# B&R Automation Studio project Soiled_PLC (part 2)

#### zzbagsfl.ab
```automation-basic
PROGRAM _CYCLIC

;----------------------------------------------------------------------
;Version 1.00 19/12/2005 D.J. First Issue - Using BAG array
;Version 2.00 24/06/2009 D.J. 32bit Cat and Cus .Cat replaced with .Prg
;Version 3.00 09/11/2009 D.J. Added Destination Counts
;----------------------------------------------------------------------
;***************************************ZEROSPOT SPECIAL*****************
Std.BagsWithDestinations 	= FALSE
Std.CustomerFound	 		   = FALSE
Std.BagsWithDestinations2  = FALSE

;Clear Destination Counts
memset(ADR(DestCountStorage),0,SIZEOF(DestCountStorage))
memset(ADR(DestCountSystem),0,SIZEOF(DestCountSystem))

LOOP CurrentLine = 1 to Std.MaxLinesBuffers DO

	LineSp = 0

	LOOP CurrentBag = Line[CurrentLine].FirstBag  TO Line[CurrentLine].LastBag DO

		EXITIF Line[CurrentLine].FirstBag = 0

		NextBag = (CurrentBag + 1)

		IF ((CurrentBag < Line[CurrentLine].LastBag) AND ((Bag[CurrentBag].Cat = 0) AND (Bag[NextBag].Cat > 0))) THEN

			;Copy Next Bag to Current
			Bag[CurrentBag]	= Bag[NextBag]
			Bag[NextBag] 	= Bag[0]

		ENDIF

		;Speed up task buy using simple variables saved 0.5ms from this task 5% CPU Usage
		CurrentDst		= Bag[CurrentBag].Dst
		IF ((CurrentDst > 0) AND (CurrentDst <= MAX_DESTINATIONS)) THEN
			IF (CurrentLine <= Std.MaxLines) THEN
				Std.BagsWithDestinations = TRUE
				DestCountStorage[CurrentDst] = DestCountStorage[CurrentDst] + 1
			ENDIF
;			DestCountSystem[CurrentDst] = DestCountSystem[CurrentDst] + 1
		ELSE IF (CurrentDst > MAX_DESTINATIONS)THEN
			Bag[CurrentBag].Dst := 0;
		ELSE IF ((CurrentDst >0) AND (CurrentDst  <= MAX_DESTINATIONS) AND (CurrentLine = 30))	THEN
			;Std.BagsWithDestinations2 = TRUE
			;DestCountStorage[CurrentDst] = DestCountStorage[CurrentDst] + 1
		ENDIF
			;FOUL LOOP bag with destination
		IF ((CurrentDst >0) AND (CurrentDst  <= MAX_DESTINATIONS) AND (CurrentLine = 30))	THEN
			Std.BagsWithDestinations2 = TRUE
			DestCountStorage[CurrentDst] = DestCountStorage[CurrentDst] + 1
		ENDIF
		;Add the line spaces up
		IF Bag[CurrentBag].Cat = 0 THEN
			LineSp = (LineSp + 1)
		ENDIF

		;For Customer FIFO table
		;-----------------------
		;Customer at front of FIFO in Storage
		;****************SPECIAL FOR ZEROSPOT*******************************
		IF ((Bag[CurrentBag].Cus = D32[401]) AND (D32[401] > 0) AND (CurrentLine <= Std.MaxLines)) THEN
			Std.CustomerFound	 	= TRUE
		ENDIF
		//Special for pairing loop, do not delete custmoer from FIFO if its on the loop
		IF ((Bag[CurrentBag].Cus = D32[401]) AND (D32[401] > 0) AND ((CurrentLine >= 30) OR (CurrentLine <= 32))) THEN
			Std.CustomerFound	 	= TRUE
		ENDIF
		IF ((Bag[259].Cus = D32[401]) AND (D32[401] > 0)) THEN
			Std.CustomerFound	 	= TRUE
		ENDIF

	ENDLOOP
	;Save the number of spaces on the current line
	Line[CurrentLine].Space = LineSp

ENDLOOP
IF (Bag[151].Cat = 0) THEN
	Line[19].Space = Line[19].Space + 1
ENDIF

IF (Bag[157].Cat = 0) THEN
	Line[19].Space = Line[19].Space + 1
ENDIF

END_PROGRAM
```

### Program Logical/Sequences/10ms/zzcp10ser (IEC, version 3.00.1)

#### zzstnser.var
```iecst
VAR
	MixProgTyp : BOOL;
	BatchFound : BOOL;
	MixCusts : BOOL;
	MixProgs : BOOL;
	MatchCust : BOOL;
	MatchBags : BOOL;
	MatchProgType : BOOL;
	MatchProg : BOOL;
	MatchCat : BOOL;
	StartPurge : BOOL;
	MixCats : BOOL;
	BankValid : BOOL;
	LineValid : BOOL;
	BagInList : ARRAY[0..30] OF BOOL;
	StartPurgeET : UDINT;
	BagNum : UINT;
	BagWgt : UINT;
	Index : UINT;
	PurgeBagsQty : UINT;
	StnNum : UINT;
	BatchCount : UINT;
	s : UINT;
	BatchWeight : UINT;
	myBag : UINT;
	r : UINT;
	MaxReverseWeight : UINT;
END_VAR
VAR RETAIN
	LineSearchManual : UINT;
END_VAR
VAR
	NumberOfPurgeBags : UINT;
	x : UINT;
END_VAR
VAR RETAIN
	SearchLine : UINT;
END_VAR
VAR
	Bank : UINT;
	Choice : UINT;
	EndofBagArray : UINT;
	PurgeBatchSize : UINT;
	MaxBatchWieght : UINT;
END_VAR
VAR RETAIN
	n : UINT;
END_VAR
VAR
	t : UINT;
	myBag_x : UINT;
	myBag_n : UINT;
END_VAR
VAR RETAIN
	SearchFound : UINT;
END_VAR
VAR
	LineSearch : ARRAY[0..4] OF UINT;
	SearchBagArray : ARRAY[0..30] OF UINT;
	PurgeBags : ARRAY[0..30] OF UINT;
	PurgeBagsInWgtOrder : ARRAY[0..30] OF UINT;
	PurgeOn : UINT;
	StatusReg : ARRAY[0..1] OF UDINT;
	SearchIndex : USINT;
	ReSearch : BOOL;
	MisMatchedLoad : BOOL;
	y : INT;
	Break : BOOL;
	StnCat : UDINT;
	GetStn : UINT;
	TestTim : BOOL;
	myStartStop : UINT;
	b : UINT;
	TON_Purge : ARRAY[0..4] OF TON_10ms;
	myBatchWgt : UDINT;
	test : UDINT;
	EmptyViking : ARRAY[0..20] OF BOOL;
	Priority : ARRAY[0..20] OF BOOL;
	E : BOOL;
	Normal : UINT;
	Over1 : UINT;
	Over2 : UINT;
	Over3 : UINT;
	Over4 : UINT;
	Viking : ARRAY[0..20] OF USINT;
	Dest : UINT;
END_VAR
```

#### zzstnser.ab
```automation-basic
;-----------------------------------------------------
;Sorting Station Search Routine - No changes required!
;-----------------------------------------------------

;----------------------------------------
;Version 1.00 19/12/2005 First Issue D.J.
;Version 2.00 03/11/2010 Revised D.J.
;Version 3.00 19/07/2016 TR... Fix bug so multiple banks can release whilst purging..
;----------------------------------------

PROGRAM _CYCLIC

IF Ldg[3].Search = 1 THEN

;Viking 5 CDC 5
IF ((Bag[80].Cat = 0) AND (Bag[81].Cat = 0) AND (Bag[82].Cat = 0)) THEN
	EmptyViking[15] = TRUE

ELSE IF ((Bag[81].Cat = 0 = 0) AND (Bag[82].Cat = 0)) THEN
	Priority[15] = TRUE

ELSE
	Priority[15]    = FALSE
	EmptyViking[15] = FALSE
ENDIF

;Viking 4 CDC 6
IF ((Bag[85].Cat = 0) AND (Bag[86].Cat = 0) AND (Bag[87].Cat = 0)) THEN
	EmptyViking[16] = TRUE

ELSE IF ((Bag[86].Cat = 0) AND (Bag[87].Cat = 0)) THEN
	Priority[16] = TRUE
ELSE
	Priority[16]    = FALSE
	EmptyViking[16] = FALSE
ENDIF

;Viking 3 CDC 7
IF ((Bag[90].Cat = 0) AND (Bag[91].Cat = 0) AND (Bag[92].Cat = 0)) THEN
	EmptyViking[16] = TRUE
ELSE IF ((Bag[91].Cat = 0) AND (Bag[92].Cat = 0)) THEN
	Priority[17] = TRUE
ELSE
	Priority[17]    = FALSE
	EmptyViking[17] = FALSE
ENDIF

;Viking 2 CDC 8
IF ((Bag[95].Cat = 0) AND (Bag[96].Cat = 0) AND (Bag[97].Cat = 0)) THEN
	EmptyViking[18] = TRUE
ELSE IF ((Bag[97].Cat = 0) AND (Bag[96].Cat = 0)) THEN
	Priority[18] = TRUE
ELSE
	Priority[18]    = FALSE
	EmptyViking[18] = FALSE
ENDIF

IF ((Bag[101].Cat = 0) AND (Bag[102].Cat = 0)AND (Bag[157].Cat = 0) AND (Bag[151].Cat = 0)) THEN
	EmptyViking[18] = TRUE
ELSE IF ((Bag[101].Cat = 0) AND (Bag[102].Cat = 0)AND (Bag[157].Cat = 0) AND (Bag[151].Cat = 0)) THEN
	Priority[19] = TRUE
ELSE
	Priority[19]    = FALSE
	EmptyViking[19] = FALSE
ENDIF

             n       = UINT(Bag[154].Cat)
      		 Normal  = (D[3000 + n]) ;destinations from cat data base
   	  		 Over1   = (D[3100 + n])
   	  		 Over2   = (D[3200 + n])
   	  		 Over3   = (D[3300 + n])
   	  		 ;Over4   = (D[2400 + n])

   	IF ((Line[Normal].SpaceBIT = 2 ) AND (D[Normal] = 1)AND (EmptyViking[Normal] = TRUE)) THEN
      	Dest = Normal
   ELSE IF ((Line[Over1].SpaceBIT = 2) AND (D[Over1] = 1 )AND (EmptyViking[Over1] = TRUE)) THEN
        Dest = Over1
   ELSE IF ((Line[Over2].SpaceBIT = 2 ) AND (D[Over2] = 1 )AND (EmptyViking[Over2] = TRUE)) THEN
        Dest = Over2
   ELSE IF ((Line[Over3].SpaceBIT = 2 ) AND (D[Over3] = 1 )AND (EmptyViking[Over3] = TRUE)) THEN
        Dest = Over3
   ;ELSE IF ((Viking[Over4] = 2 ) AND (D[Over4 ] = 1 )AND (EmptyViking[Over4] = TRUE)) THEN
    ;    Dest = Over4

   ELSE IF ((Line[Normal].SpaceBIT = 2 ) AND (D[Normal] = 1)AND (Priority[Normal] = TRUE)) THEN
      	Dest = Normal
   ELSE IF ((Line[Over1].SpaceBIT = 2) AND (D[Over1] = 1 )AND (Priority[Over1] = TRUE)) THEN
        Dest = Over1
   ELSE IF ((Line[Over2].SpaceBIT = 2 ) AND (D[Over2] = 1 )AND (Priority[Over2] = TRUE)) THEN
        Dest = Over2
   ELSE IF ((Line[Over3].SpaceBIT = 2 ) AND (D[Over3] = 1 )AND (Priority[Over3] = TRUE)) THEN
        Dest = Over3
   ;ELSE IF ((Viking[Over4] = 2 ) AND (D[Over4 + 7] = 1 )AND (Priority[Over4] = TRUE)) THEN
   ;     Dest = Over4
    ELSE IF ((Line[Normal].SpaceBIT > 0 ) AND (D[Normal ] = 1)) THEN
       Dest = Normal
    ELSE IF ((Line[Over1].SpaceBIT > 0) AND (D[Over1] = 1 )) THEN
        Dest = Over1
   ELSE IF ((Line[Over2].SpaceBIT > 0 ) AND (D[Over2] = 1 )) THEN
        Dest = Over2
   ELSE IF ((Line[Over3].SpaceBIT > 0 ) AND (D[Over3] = 1 )) THEN
        Dest = Over3
   ;ELSE IF ((Viking[Over4] > 0 ) AND (D[Over4 + 7] = 1 )) THEN
   ;     Dest = Over4
   ENDIF

  IF ((Dest > 0) AND (Bag[154].Dst = 0) AND (Line[Dest].SpaceBIT>0)) THEN
  	Ldg[3].Search = 2
  	Ldg[3].Found       = Dest
  ELSE IF (Bag[154].Dst > 14)AND (Line[Bag[154].Dst].SpaceBIT>0) THEN
  	Ldg[3].Search = 2
  	Ldg[3].Found       = Bag[154].Dst
 ENDIF
ENDIF
Debug:

END_PROGRAM
```

### Program Logical/Sequences/10ms/zzBITcal (IEC) - * Bags In Transit Calculation

#### zzbitcal.var
```iecst
VAR RETAIN
	TotalTransitBags : UINT;
	n : UINT;
	BITDest : ARRAY[0..199] OF UINT;
	Destination : USINT;
	SpaceBIT : ARRAY[0..199] OF UINT;
	Spaces : INT;
END_VAR
VAR
	BITBag : UINT;
	ArraySize : UINT;
	Error : UINT;
	BoostSD4 : BOOL;
	BoostSDC4 : BOOL;
	BoostSDC5 : BOOL;
	lineValid : BOOL;
END_VAR
```

#### zzbitcal.ab
```automation-basic
PROGRAM _INIT

BITBag 	= 2
Error 	= 0
;Transfer Belt Bags
;LOOP n = 1 TO 2 DO
	;BITDest[1] = 153
	;BITDest[2] = 152
	;BITDest[3] = 151
	;BITDest[4] = 157
;	BITDest[BITBag] = n
;	BITBag = BITBag + 1
;ENDLOOP

;Bags in transit
LOOP n = 110 TO 164 DO

	ArraySize = (SIZEOF(BITDest) / 2)
	IF (BITBag <= ArraySize) THEN
		BITDest[BITBag] = n
		BITBag = BITBag + 1
	ELSE
		Error = 1
	ENDIF
ENDLOOP

TotalTransitBags = (BITBag - 1)
END_PROGRAM

PROGRAM _CYCLIC
	(* cyclic program *)

	;-----------------------------------------------------------
	;Revision 1.00 19/12/2005 D.J. First Issue - Using BAG array
	;-----------------------------------------------------------

	;Find the Space on each Storage line including the Ongoing and Offgoing Bags In Transit

	;See Init Routine - Change settings for bags in transit bag numbers

	;Clear local calculation
	LOOP n = 1 TO Std.MaxLinesBuffers DO
		SpaceBIT[n] = 0
	ENDLOOP

	memset(ADR(DestCountArea1),0,SIZEOF(DestCountArea1))

	;Ensure the destination is less than the Array size of SpaceBIT	(normally 100)
	LOOP n = 1 TO TotalTransitBags DO
	;LOOP n = 3 TO 3 DO
		Destination = Bag[BITDest[n]].Dst

		lineValid = ((Destination <= Line[Destination].FirstBag) OR (Destination > Line[Destination].LastBag));//Stop bit being counted twice if on own line.
		IF lineValid AND (Destination > 0) AND (Destination < 15)  THEN
			SpaceBIT[Destination] = SpaceBIT[Destination] + 1
			DestCountSystem[Destination] = DestCountSystem[Destination] + 1
		ENDIF
	ENDLOOP
	IF (Bag[153].Cat > 0) AND (Bag[153].Dst>0) THEN
			SpaceBIT[Bag[153].Dst] = SpaceBIT[Bag[153].Dst] + 1
			DestCountSystem[Bag[153].Dst] = DestCountSystem[Bag[153].Dst] + 1
	ENDIF
	IF (Bag[152].Cat > 0) AND (Bag[152].Dst>0) THEN
			SpaceBIT[Bag[152].Dst] = SpaceBIT[Bag[152].Dst] + 1
			DestCountSystem[Bag[152].Dst] = DestCountSystem[Bag[152].Dst] + 1
	ENDIF
	IF (Bag[166].Cat > 0) AND (Bag[166].Dst>0) THEN
			SpaceBIT[Bag[166].Dst] = SpaceBIT[Bag[166].Dst] + 1
			DestCountSystem[Bag[166].Dst] = DestCountSystem[Bag[166].Dst] + 1
	ENDIF
	IF (Bag[151].Cat > 0) AND (Bag[151].Dst>0) THEN
			SpaceBIT[Bag[151].Dst] = SpaceBIT[Bag[151].Dst] + 1
			DestCountSystem[Bag[151].Dst] = DestCountSystem[Bag[151].Dst] + 1
	ENDIF
	IF (Bag[157].Cat > 0) AND (Bag[157].Dst>0) THEN
			SpaceBIT[Bag[157].Dst] = SpaceBIT[Bag[157].Dst] + 1
			DestCountSystem[Bag[157].Dst] = DestCountSystem[Bag[157].Dst] + 1
	ENDIF
	;Once all calculated then update the global line space
	LOOP n = 1 TO Std.MaxLinesBuffers DO
	;LOOP n = 1 TO 1 DO
		Spaces = (INT(Line[n].Space) - INT(SpaceBIT[n]))
		IF Spaces > 0 THEN
			Line[n].SpaceBIT = UINT(Spaces)
		ELSE
			Line[n].SpaceBIT = 0
		ENDIF
	ENDLOOP

END_PROGRAM
```

### Program Logical/Sequences/10ms/zzCusFIFO (IEC) - * Customer FIFO 

#### zcusfifo.var
```iecst
VAR RETAIN
	OngoingCus : UDINT;
	EditCus : UDINT;
	n : UDINT;
	x : UINT;
END_VAR
VAR
	myBag : UINT;
	InsDel : DINT;
	InsPos : UDINT;
	DelPos : UDINT;
END_VAR
```

#### zcusfifo.ab
```automation-basic
PROGRAM _CYCLIC
;------------------------------------------------------
;Revision 1.00 11/02/2002 D.J. First Issue
;Revision 2.00 11/06/2002 D.J. Included Bags In Transit
;------------------------------------------------------

;Include any Bags In Transit if required

;New Customers
InsPos		= D32[496]
DelPos		= D32[497]
OngoingCus 	= D32[498]
EditCus		= D32[499]

IF Std.CustomerFIFO THEN

	;The following are Set by the "Bag Shuffle"
	;First customer not found clear from the FIFO
	IF NOT Std.CustomerFound THEN
		D32[401] = 0
	ENDIF

	;Shuffle the Table down
	D32[400] = 0

	LOOP n = 401 TO 494 DO

		IF ((D32[n] = 0) AND (D32[n + 1] > 0)) THEN
			D32[n] = D32[n + 1]
			D32[n + 1] = 0
		ENDIF

		IF (D32[n] > 0) THEN
			;Inc FIFO Header Count
			D32[400] = (D32[400] + 1)
		ENDIF

		;Clear New Customer if found
		IF ((OngoingCus > 0) AND (OngoingCus = D32[n])) THEN
			OngoingCus = 0
		ENDIF

		;Clear Edited Customer if found
		IF ((EditCus > 0) AND (EditCus = D32[n])) THEN
			EditCus = 0
		ENDIF

	ENDLOOP

	;Insert From TrackView
	IF ((InsPos > 0) AND (EditCus > 0)) THEN
		LOOP n = 495 DOWNTO (400 + InsPos) DO
			D32[n] = D32[n - 1]
		ENDLOOP
		D32[400 + InsPos] 	= EditCus
		InsPos 				= 0
		EditCus				= 0
	ENDIF

	;Delets From TrackView
	IF (DelPos > 0) THEN
		D32[400 + DelPos] 	= 0
		DelPos 				= 0
	ENDIF

	;D32[498] = Ongoing New Customer
	IF ((OngoingCus > 0) AND (D32[401 + D32[400]] = 0)) THEN
		D32[401 + D32[400]]	= OngoingCus
		OngoingCus 			= 0
		D32[400] 			= (D32[400] + 1)
	ENDIF

	;D32[499] = Edited New Customer
	IF ((EditCus > 0) AND (D32[401 + D32[400]] = 0)) THEN
		D32[401 + D32[400]]	= EditCus
		EditCus 			= 0
		D32[400] 			= (D32[400] + 1)
	ENDIF

	;Find the Current Customer for each Discharger and allocate the Next Customer

	LOOP x = 1 TO Std.MaxDischargers DO

		Uld[x].FIFONextCustomer = 0
		Uld[x].FIFOCustomerFound = FALSE

		;If No Customer then Allocate with the First
		IF (Uld[x].FIFOCustomer = 0) THEN
			Uld[x].FIFOCustomer = D32[401]
		ENDIF

		;If Next Customer available then allocate New Customer
		IF (D32[400] > 0) THEN
			LOOP n = 401 TO (D32[400] + 400) DO
				IF ((Uld[x].FIFOCustomer = D32[n]) AND (D32[n] > 0)) THEN
					Uld[x].FIFOCustomerFound = TRUE
					IF (D32[n + 1] > 0) THEN
						Uld[x].FIFONextCustomer = D32[n + 1]
					ENDIF
				ENDIF
			ENDLOOP
		ENDIF

		;If the current customer has been removed then set the next as the first
		IF ((Uld[x].FIFONextCustomer = 0) AND NOT Uld[x].FIFOCustomerFound) THEN
			Uld[x].FIFONextCustomer = D32[401]
		ENDIF

	ENDLOOP

ENDIF

D32[496] = InsPos
D32[497] = DelPos
D32[498] = OngoingCus
D32[499] = EditCus
END_PROGRAM
```

- Program Logical/Sequences/10ms/zzCount (IEC) - Counting frames inputs & Piece Weights (no source held here)

### Program Logical/Sequences/10ms/zzStnMix (IEC)

#### zzstnmix.ab
```automation-basic
PROGRAM _CYCLIC
;----------------------
;Sorting Station Mixing
;----------------------

;----------------------------------------
;Version 1.00 09/12/2005 D.J. First Issue
;----------------------------------------

;Notes:
;When the operator changes either the Category or Customer of any station then the report should be written.
;If the Customer or Category is set to zero the report will be written for the previous Cat and Cus however
;the previous Cat and Cus will be set to zero. When the Cat or Cus is next changed there will be no report

IF Std.StationReports THEN

	;Special for Mewa only box 1 to 6 are reported on
	LOOP n = 1 TO Std.MaxWeighstations DO

		StnBag = LDG_GetBagFromStation(Std.StationBagsStart,n);n + (Std.StationBagsStart[1] - 1) ;Assumes all station bags will follow in order

		IF (ReportLoading[n].Cat = 0) THEN

			;Check if Category or Customer have been changed
			CatChanged 	= (Bag[StnBag].Cat <> StnPrev[n].Cat)
			CatValid   	= (StnPrev[n].Cat > 0)

			CusChanged 	= (Bag[StnBag].Cus <> StnPrev[n].Cus)
			CusValid   	= (StnPrev[n].Cus > 0)

			;Check if anything has been added and current weight is not less than the previous
			WgtValue 	= Stn[n].Weight	- INT(StnPrev[n].Wgt)
			WgtValid 	= (WgtValue > 0)

			;Check if anything has been added and current weight is not less than the previous
			CntValue 	= Stn[n].Count - INT(StnPrev[n].Cnt)
			CntValid 	= (CntValue > 0)

			;Ensure valid values as we report on either a weight or count change
			IF (WgtValue < 0) THEN
				WgtValue = 0
			ENDIF

			IF (CntValue < 0) THEN
				CntValue = 0
			ENDIF

			IF ((CatChanged OR CusChanged) AND CusValid AND CatValid AND (WgtValid OR CntValid)) THEN

				ReportLoading[n].Prg = StnPrev[n].Prg		;Program
				ReportLoading[n].Cat = StnPrev[n].Cat		;Category
				ReportLoading[n].Cus = StnPrev[n].Cus		;Customer
				ReportLoading[n].Wgt = UINT(WgtValue)		;Weight
				ReportLoading[n].Cnt = UINT(CntValue)		;Count
				ReportLoading[n].Stn = n         			;Station
				ReportLoading[n].Mcn = 0					;Machine
				ReportLoading[n].Bid = StnPrev[n].Bid		;Bag ID
				ReportLoading[n].Mis = n
				ReportLoading[n].Act = repMix
				ReportLoading[n].Ur1 = 0
				ReportLoading[n].Ur2 = 0
				ReportLoading[n].Rkg = 0

			ENDIF

			;Set Previous to Current even if the Previous values were not valid
			IF (CatChanged OR CusChanged) THEN
				StnPrev[n].Prg = Bag[StnBag].Prg
				StnPrev[n].Cat = Bag[StnBag].Cat
				StnPrev[n].Cus = Bag[StnBag].Cus
				StnPrev[n].Wgt = Stn[n].Weight
				StnPrev[n].Cnt = Stn[n].Count
				StnPrev[n].Bid = Bag[StnBag].Bid
			ENDIF

		ENDIF

	ENDLOOP

ENDIF

END_PROGRAM
```

### Program Logical/Sequences/10ms/4_spn1_ref (IEC, version 1.00.0) - *REF ONLY

#### 4_spn1Cyclic.ab
```automation-basic
PROGRAM _CYCLIC
; 	(* cyclic program *)

;Sequence 4 - Ongoing To Storage D[904]

;-----------------------------------------
;Revision 1.00 09/12/2005 D.J. First Issue
;-----------------------------------------

;Inputs
OnGoingEnable 		= ((D[14] > 0) AND NOT Std.HaltSys)

I_BagatBuffer[1]	= Request.VC[1] ;X[7].X13
;I_BagatBuffer[2]	= FALSE
;I_BagatBuffer[3]	= FALSE
;I_BagatBuffer[4]	= FALSE

O_Reset 		  	= FALSE
O_OpenSelect[1]		= FALSE
;O_OpenSelect[2]	= FALSE
;O_OpenSelect[3]	= FALSE
;O_OpenSelect[4]	= FALSE

Enable.PN[1]		= FALSE

Alarm[4].Name 		= 0
Alarm[4].Bag		= 224
Alarm[4].Beacon		= TRUE
Alarm[4].Extra	 	= 0
Alarm[4].Time		= 3000

;Setup Sequence
;--------------
STEP = D[904]
;Setup Pulse contact
PLS = (STEP <> LASTSTEP)
LASTSTEP = STEP

;Check if Recirculation bag needs a destination
;IF ((Bag[107].Cat > 0) AND (Bag[107].Dst = 0) AND (D[1005] > 0) AND (D[1005] <= 6) AND (D[1006] > 0)) THEN
;	Bag[107].Dst 	= D[1005]
;	D[1006] 		= (D[1006] - 1)
;ENDIF

;Step 0 - Disabled
IF (STEP = 0) THEN
	;Disabled
ENDIF

;Step 1 - Reset Ongoing Points
TON_10ms((STEP = 1),300,ResetPoints,ResetPointsET)
IF (STEP = 1) THEN
	Dest  	= 0
	Buff 	= 0
	O_Reset = NOT ResetPoints
	IF (ResetPoints AND OnGoingEnable) THEN
		D[904] = 2
	ENDIF
ENDIF

;Set Max Buffers to search
MaxBuffers = 1

;Bag Settles at each buffer
;TON_10ms(I_BagatBuffer[1],300,SettledBuffer[1],SettledBufferET[1])
SettledBuffer[1] = I_BagatBuffer[1] ;SVC1
;TON_10ms(I_BagatBuffer[2],300,SettledBuffer[2],SettledBufferET[2])

BufferBagNum[1]		= 222
;BufferBagNum[2]	= 250

;Step 2 - Search for a valid Bag at one of the buffers
IF (STEP = 2) THEN

	Buff 	= 0
	Dest 	= 0

	IF OnGoingEnable THEN

		Alarm[4].Name 	= almNoAlarm
		Alarm[4].Time	= 2000

		LOOP Bfr = 1 TO MaxBuffers DO

			;Set Test Value for Monitoring
			IF TestBuffer > 0 THEN
				Buffer = TestBuffer
			ELSE
				Buffer = Bfr
			ENDIF

			BufferBag		= BufferBagNum[Buffer]
			BufferSettled 	= SettledBuffer[Buffer]
			BufferCat 		= Bag[BufferBag].Cat
			BufferDst 		= Bag[BufferBag].Dst

			DestValid = ((BufferDst >= 1) AND (BufferDst <= Std.MaxLines))

			IF (BufferSettled AND (BufferCat > 0) AND DestValid AND (Bag[224].Cat = 0)) THEN
				n = BufferDst
				IF ((Line[n].Space > 0) AND Line[n].Clear) THEN
					Dest = n
					Buff = Buffer
					;IF (Buffer = 1) THEN
						D[904] 	= 3
					;ELSE
					;	D[904]  = 4
					;ENDIF
				ELSE
					Alarm[4].Name 	= almDestinationNotValid
					Alarm[4].Bag	= BufferBag
				ENDIF
			ENDIF

			;Buffer Alarms
			;IF (BufferCat > 0) AND NOT BufferSettled THEN
			;	Alarm[4].Name 	= almBagNotAtProx
			;	Alarm[4].Bag	= BufferBag
			;ELSE IF (BufferCat = 0) AND BufferSettled THEN
			;	Alarm[4].Name 	= almBagNotShownOnScreen
			;	Alarm[4].Bag	= BufferBag
			;ENDIF

		ENDLOOP

	ENDIF

ENDIF

;Clear Line Selections
LOOP n = 1 TO Std.MaxLines DO
	LineSelect[n] = FALSE
ENDLOOP

;Step 3 - Enable VC1 to Release a bag
IF (STEP = 3) THEN
	Enable.PN[1] = TRUE

	IF PLS THEN
		C[Dest] = 0
	ENDIF

	LineSelect[Dest] = TRUE
	IF NOT Request.VC[1] THEN
		D[904] = 4
	ENDIF
ENDIF

;Step 4 - Select line / open buffer stop
IF (STEP = 4) THEN

	LineSelect[Dest] 	= TRUE
	O_OpenSelect[Buff] 	= TRUE

	IF PLS THEN
		;C[Dest] = 0
		IF (Bag[224].Cat = 0) AND (Bag[BufferBagNum[Buff]].Cat > 0) THEN
			Bag[224]				 	= Bag[BufferBagNum[Buff]]
			Bag[BufferBagNum[Buff]]	 	= Bag[0]
		ENDIF
	ENDIF

	;Bag arrived on selected line
	IF Line[Dest].Trip THEN
		D32[498] 						= Bag[224].Cus	;Set Customer for Customer FIFO
		Bag[224].Dst 				= 0 		    ;Clear Destination
		Bag[Line[Dest].LastBag] 	= Bag[224]
		Bag[224] 					= Bag[0]
		D[904] 						= 1
	ENDIF

	Alarm[4].Name = almBagNotArrived

ENDIF

;Alarms
TimerAlarm.IN = NOT PLS AND (Alarm[4].Name > 0) AND (AlarmOld = Alarm[4].Name)
TimerAlarm.PT = Alarm[4].Time
TimerAlarm FUB TON_10ms()
Alarm[4].On = TimerAlarm.Q
Alarm[4].ET = TimerAlarm.ET

AlarmOld = Alarm[4].Name ;Need to ensure alarm changes as may be multiple alarms on step 2

;Outputs
Y[4].Y01 = LineSelect[1] OR LineSelect[2]
Y[4].Y02 = LineSelect[3]
Y[4].Y03 = LineSelect[3]
Y[4].Y04 = LineSelect[4]
Y[4].Y05 = LineSelect[5]
Y[4].Y06 = LineSelect[6]
Y[4].Y07 = LineSelect[7]
Y[4].Y08 = LineSelect[8]
Y[4].Y09 = LineSelect[9]
Y[4].Y10 = LineSelect[10]
Y[4].Y11 = LineSelect[11]
Y[4].Y12 = LineSelect[12]
Y[4].Y13 = LineSelect[13]
Y[4].Y14 = LineSelect[14] OR O_Reset

Y[3].Y15 = LineSelect[1]
Y[3].Y14 = LineSelect[2]

END_PROGRAM
```

#### 4_spn1.var
```iecst
VAR RETAIN
	n : UINT;
	STEP : UINT;
	ResetPointsET : TIME;
	ResetPoints : BOOL;
	LASTSTEP : UINT;
	PLS : BOOL;
	LineSelect : ARRAY[0..19] OF BOOL;
	OnGoingEnable : BOOL;
	O_Reset : BOOL;
	I_BagatBuffer : ARRAY[0..4] OF BOOL;
END_VAR
VAR
	SettledBuffer : ARRAY[0..4] OF BOOL;
	Buffer : UINT;
	AlarmOld : UINT;
	BufferBag : UINT;
	DestValid : BOOL;
	Dest : UINT;
	BufferDst : UINT;
	BufferBagNum : ARRAY[0..4] OF UINT;
	TestBuffer : UINT;
	TimerAlarm : TON_10ms;
	Bfr : UINT;
	BufferSettled : BOOL;
	BufferCat : UDINT;
	MaxBuffers : UINT;
	Buff : UINT;
	O_OpenSelect : ARRAY[0..4] OF BOOL;
END_VAR
```

### Program Logical/Sequences/10ms/1_stnsa_ref (IEC) - *FROM OLD PROGRAM REF ONLY

#### 1_stnsa.var
```iecst
VAR RETAIN
	n : UINT;
	OpenBag : ARRAY[0..99] OF BOOL;
	STEP : UINT;
	PLS : ARRAY[0..99] OF BOOL;
	LASTSTEP : ARRAY[0..99] OF UINT;
	BagClosed : ARRAY[0..99] OF BOOL;
	BagClosedET : ARRAY[0..99] OF TIME;
	OpenTime : UINT;
	BagOpenedET : ARRAY[0..99] OF TIME;
	BagOpened : ARRAY[0..99] OF BOOL;
	CloseTime : UINT;
END_VAR
VAR
	Bank : UINT;
	TimerOpen : ARRAY[0..49] OF TON_10ms;
	TimerClosed : ARRAY[0..49] OF TON_10ms;
	TimerAlarm : ARRAY[0..49] OF TON_10ms;
	StnBag : UINT;
	x : INT;
END_VAR
```

#### 1_stnsaCyclic.ab
```automation-basic
PROGRAM _CYCLIC
	(* cyclic program *)

;Honeycombe Sorting Station Control
;----------------------------------------------------
;Revision 1.00 10/01/2002 D.J. First Issue
;Revision 2.00 07/02/2005 D.J. Removed Stn Mix
;Revision 3.00 22/08/2006 D.J. Changed to timer array
;----------------------------------------------------

Bank = 1

;Timers
OpenTime  = 700
CloseTime = 300

LOOP x = 1 TO Ldg[Bank].NoStations DO
	n = Ldg[Bank].Stations[x]

	;Bag open timers
	TimerOpen[n].IN 	= OpenBag[n]
	TimerOpen[n].PT		= OpenTime
	TimerOpen[n] FUB TON_10ms()

	BagOpened[n] 		= TimerOpen[n].Q
	BagOpenedET[n]		= TimerOpen[n].ET

	;Bag closed timers
	TimerClosed[n].IN 	= NOT OpenBag[n]
	TimerClosed[n].PT	= CloseTime
	TimerClosed[n] FUB TON_10ms()

	BagClosed[n] 		= TimerClosed[n].Q
	BagClosedET[n]		= TimerClosed[n].ET

	;Update bag weight
	//StnBag = n + (Std.StationBagsStart[Bank] - 1)
	StnBag = LDG_GetBagFromStation(Std.StationBagsStart,n);
	Bag[StnBag].Wgt = Stn[n].Weight
	Bag[StnBag].Cnt = Stn[n].Count

	Alarm[40 + n].Name 		= 0
	Alarm[40 + n].Bag		= StnBag
	Alarm[40 + n].Beacon	= TRUE
	Alarm[40 + n].Extra		= 0
	Alarm[40 + n].Time		= 2000

	Stn[n].LampOn 		= FALSE

	STEP = D[940 + n]
	;Setup Pulse contact
	PLS[n] = (STEP <> LASTSTEP[n])
	LASTSTEP[n] = STEP

	;Step 0 - Disabled
	IF (STEP = 0) THEN
		Stn[n].LampOn = TRUE
		;Disabled
	ENDIF

	IF (STEP = 1) THEN
		Stn[n].LampOn = TRUE
		IF D[901] = n THEN
			D[901] = 0
		ENDIF
		IF BagClosed[n] THEN
			D[940 + n] = 2
		ENDIF
		Alarm[40 + n].Name = almStationNotClosed
	ENDIF

	IF (STEP = 2) THEN
		Stn[n].LampOn = ((Stn[n].SP1 AND Std.Clock2s) OR Stn[n].SP2 OR (Stn[n].SP3 AND Std.Clock200ms))
		IF ((D[901] = n) AND Ldg[Bank].EnableStnRelease) THEN
			D[940 + n] = 3
		ENDIF
		IF ((Bag[StnBag].Cat > 0) AND Stn[n].SP3) THEN
			Alarm[40 + n].Name = almBagOverWeight
		ENDIF
	ENDIF

	IF (STEP = 3) THEN
		Stn[n].LampOn = TRUE
		IF (BagOpened[n] AND ((Stn[n].Weight < 30) OR Test.Stations) AND Ldg[Bank].BeltHasRun) THEN
			Stn[n].QTime 	= 0
			D[940 + n] 		= 1
		ENDIF
		IF (Stn[n].Weight >= 30) THEN
			Alarm[40 + n].Name = almStationNotEmpty
		ENDIF
	ENDIF

	OpenBag[n] = (STEP = 3)

	;Alarm timer
	TimerAlarm[n].IN 	= NOT PLS[n] AND (Alarm[40 + n].Name > 0)
	TimerAlarm[n].PT	= Alarm[40 + n].Time
	TimerAlarm[n] FUB TON_10ms()

	Alarm[40 + n].ET	= TimerAlarm[n].ET
	Alarm[40 + n].On 	= TimerAlarm[n].Q

ENDLOOP

;Outputs
;-------

Y[31].Y05 = OpenBag[1]
Y[31].Y06 = OpenBag[2]
Y[31].Y07 = OpenBag[3]
Y[31].Y08 = OpenBag[4]
Y[31].Y13 = OpenBag[5]
Y[31].Y14 = OpenBag[6]
Y[31].Y15 = OpenBag[7]
Y[31].Y16 = OpenBag[8]
Y[32].Y05 = OpenBag[9]
Y[32].Y06 = OpenBag[10]
Y[32].Y07 = OpenBag[11]
Y[32].Y08 = OpenBag[12]
Y[32].Y13 = OpenBag[13]
Y[32].Y14 = OpenBag[14]
Y[32].Y15 = OpenBag[15]
Y[32].Y16 = OpenBag[16]

Y[31].Y01 = Stn[1].LampOn
Y[31].Y02 = Stn[2].LampOn
Y[31].Y03 = Stn[3].LampOn
Y[31].Y04 = Stn[4].LampOn
Y[31].Y09 = Stn[5].LampOn
Y[31].Y10 = Stn[6].LampOn
Y[31].Y11 = Stn[7].LampOn
Y[31].Y12 = Stn[8].LampOn
Y[32].Y01 = Stn[9].LampOn
Y[32].Y02 = Stn[10].LampOn
Y[32].Y03 = Stn[11].LampOn
Y[32].Y04 = Stn[12].LampOn
Y[32].Y09 = Stn[13].LampOn
Y[32].Y10 = Stn[14].LampOn
Y[32].Y11 = Stn[15].LampOn
Y[32].Y12 = Stn[16].LampOn
END_PROGRAM
```

### Program Logical/Sequences/10ms/2_stb1 (IEC) - *For Reference only-- Adjust as required.

#### beltCyclic.ab
```automation-basic
PROGRAM _INIT
	_setBeltTime

END_PROGRAM

PROGRAM _CYCLIC
 	(* cyclic program *)

;Sequence 2 - Transfer Belt 1 from Stations 1-8

;-----------------------------------------
;Revision 1.00 18/01/2006 D.J. First Issue
;-----------------------------------------

;Inputs and Outputs
;-----------------

myBank 			= 1
myBelt			= 1
mySeq			= 2
myBag			= 163
myOutBag		= 161
myZone			= 0

MixCats			= (D[369] > 0)
MixCusts		= (D[366] > 0)	;Allow mixing of customers?
MixProgs		= (D[367] > 0)	;Allow mixing of Programs?

;I_PhotoBottom		      	= X[3].X08
I_PhotoTop   		      	= X[3].X07
I_Manual_Stop               = X[15].X08
I_PhotoReverse            	= FALSE
I_InvStatus					= TRUE

;Belt add times in an array for each station as station number will not work..
;LOOP n = 20 DOWNTO 1 DO
;	BeltAddTimeArray[n]		= n
;ENDLOOP

RequestRel.TransferBelt[myBelt]		  	= FALSE
Request.TransferBelt[myBelt]		    = FALSE

O_RunBelt 					= FALSE
O_Reverse					= FALSE
O_SlowBelt					= FALSE

;Check all stations are closed.
StationOpen = FALSE
LOOP n = 1 TO Ldg[myBank].NoStations DO
	stnNo = Ldg[myBank].Stations[n]
	IF (D[950 + stnNo] = 3) THEN
		StationOpen = TRUE
	ENDIF
ENDLOOP

Alarm[mySeq].Name 				= 0
Alarm[mySeq].Bag				= myBag
Alarm[mySeq].Beacon				= FALSE
Alarm[mySeq].Extra				= 0
Alarm[mySeq].Time			  	= 5000

n = D[900 + Std.StationBankReg + myBank] ;Selected Station

STEP = D[900 + mySeq]
;Setup Pulse contact
PLS = (STEP <> LASTSTEP)
LASTSTEP = STEP

;Step 0 - Disabled
IF STEP = 0 THEN
	;Disabled
ENDIF

;Step 1 - Check no stations are releasing
IF STEP = 1 THEN
	;Don't allow stations to release
	Ldg[myBank].EnableStnRelease = FALSE
	Std.PurgeBank[myBank].PurgeOn = 0 ; Clear to display Purge
	Std.PurgeBank[myBank].StationsStatus[0] = 0 ;trackview TO display Purge
	Std.PurgeBank[myBank].StationsStatus[1] = 0
	;No Station Releaseng and switched on
	IF (NOT StationOpen AND (D[mySeq] > 0) AND NOT I_Manual_Stop) THEN
		IF (Bag[myBag].Cat = 0) THEN
			D[900 + mySeq] = 2 ;No Bag on belt
		ELSE
			D[900 + mySeq] = 4 ;Bag on belt
		ENDIF
	ENDIF
	Alarm[mySeq].Name = almNoAlarm
ENDIF

;Step 2 - Enable Station search
IF STEP = 2 THEN
	IF (Bag[myBag].Cat > 0) THEN
;		D[900 + mySeq] = 4
	ENDIF
	;Check each station to see if a manual destination has been set
	LOOP n = 1 to Ldg[myBank].NoStations DO

		//StnBag = Std.StationBagsStart + Ldg[myBank].Stations[n] - 1
		StnBag = LDG_GetBagFromStation(Std.StationBagsStart,n)

		IF ((Bag[StnBag].Dst > 0) AND (Bag[StnBag].Dst < 99) AND (D[mySeq] > 0)) THEN ;Dest 99 = Empty Bag in station
			Stn[n].DestManual = Bag[StnBag].Dst
		ELSE
			Stn[n].DestManual = 0
		ENDIF
		;For pairing set number of spaces to search for
		Stn[n].SpacesRequired = 1 ;D[2000 + Bag[StnBag].Prg]

	ENDLOOP

	;Station Search

	IF ((Ldg[myBank].Search = 0) AND (D[mySeq] > 0) AND NOT Std.HaltSysZone[myZone] AND EnableRel.TransferBelt[myBelt])  THEN
		Ldg[myBank].Search = 1
		PurgeBagIndex = 0
	ELSE IF ((Ldg[myBank].Search = 2) AND (Ldg[myBank].Found > 0)) THEN ;
		IF (Ldg[myBank].Found < 97) THEN
			D[900 + Std.StationBankReg + myBank] 	= Ldg[myBank].Found
			n 	= D[900 + Std.StationBankReg + myBank]
;		ELSE IF (Ldg[myBank].Found = 98) OR (Ldg[myBank].Found = 97) THEN ; Reverse belt
;			D[900 + mySeq] = 9
;			GOTO ExitStep2 ; Ignore the rest of Step 2
		ELSE
;			IF (Ldg[myBank].Found = 98) OR (Ldg[myBank].Found = 97) THEN
;				Ldg[myBank].Line = 21 ; Set Destination to SDC1
;			ENDIF
		;	Purge = TRUE

			n = LDG_GetStationFromBag(Std.StationBagsStart,Std.PurgeBank[myBank].PurgeBatch[PurgeBagIndex])
			IF (n = 0) OR (n > Ldg[myBank].Stations[Ldg[myBank].NoStations]) THEN
				Ldg[myBank].Search = 0
				GOTO ExitStep2
			ENDIF
			D[900 + Std.StationBankReg + myBank] = n
			Std.PurgeBank[myBank].PurgeOn = 1 ; Send to trackview to display Purge
			myStnReg = (n > 32)
			IF (myStnReg = 0)THEN
				myStnBit =	n - 1
			ELSE IF (myStnReg = 1)THEN
				myStnBit = 	n - 33
				ELSE
				myStnBit = 0
			ENDIF
			Std.PurgeBank[myBank].StationsStatus[myStnReg] = BIT_SET(Std.PurgeBank[myBank].StationsStatus[myStnReg],myStnBit)
			;Get highest belt add time... Use array as station numbers are opposite to distanct
			IF BeltAddTimeArray[n] > BeltAddTime THEN
				BeltAddTime = BeltAddTimeArray[n]
			ENDIF
		ENDIF
		StnBag = LDG_GetBagFromStation(Std.StationBagsStart,n)
		;Clear the release button count if used
		Stn[n].ManualRelease 	= FALSE
		Stn[n].Purge 			= FALSE
		Stn[n].PurgeReverse	 	= FALSE
		Stn[n].PBCount 			= 0
		;------Write Report------
	;	IF Std.StationReports AND (Ldg[myBank].Found <> 98) AND (Ldg[myBank].Found <> 97)THEN
        IF Std.StationReports THEN
			IF (ReportLoading[n].Cat = 0)  THEN
				IF Purge THEN
					IF (PurgeBagIndex < Std.PurgeBank[myBank].PurgeBagQty) THEN
						PurgeBagIndex = PurgeBagIndex + 1
					ENDIF
				ENDIF
				WeightValue = Stn[n].Weight - INT(StnPrev[n].Wgt)
				WeightValid = (WeightValue > 0)

				;Check if anything has been added and current weight is not less than the previous
				CountValue = Stn[n].Count - INT(StnPrev[n].Cnt)
				CountValid = (CountValue > 0)
				IF (WeightValid OR CountValid) THEN
					;Ensure valid values as we report on either a weight or count change
					IF (WeightValue < 0) THEN
						WeightValue = 0
					ENDIF

					IF (CountValue < 0) THEN
						CountValue = 0
					ENDIF
					myTimeStamp = CurrentTimestamp
					ReportLoading[n].Prg = Bag[StnBag].Prg 			;Program
					ReportLoading[n].Cat = Bag[StnBag].Cat			;Category
					ReportLoading[n].Cus = Bag[StnBag].Cus			;Customer
					ReportLoading[n].Wgt = UINT(WeightValue)		;Weight
					ReportLoading[n].Cnt = UINT(CountValue)			;Count
					ReportLoading[n].Stn = n         				;Station
					ReportLoading[n].Mcn = 0						;Machine
					ReportLoading[n].Bid = Bag[StnBag].Bid			;Batch ID
					ReportLoading[n].TimeStamp = myTimeStamp

				ENDIF
			ENDIF
		ELSE
			myTimeStamp = CurrentTimestamp
			IF Purge THEN
				IF (PurgeBagIndex < Std.PurgeBank[myBank].PurgeBagQty) THEN
					PurgeBagIndex = PurgeBagIndex + 1
				ENDIF
			ENDIF
		ENDIF

		;Set Previous Cat and Cus to Current and Clear Weight and Count
		StnPrev[n].Prg 	= Bag[StnBag].Prg
		StnPrev[n].Cat 	= Bag[StnBag].Cat
		StnPrev[n].Cus 	= Bag[StnBag].Cus
		StnPrev[n].Wgt 	= 0
		StnPrev[n].Cnt 	= 0
		StnPrev[n].Bid 	= Bag[StnBag].Bid

		Ldg[myBank].EnableStnRelease = TRUE
		;Clear Manual Release and Count
		Stn[n].ManualRelease 	= FALSE
		Stn[n].Count			= 0
		BeltAddTime = BeltAddTimeArray[n]
		;Keep A record of purged bags to attach the data for the biggest loads
		IF Purge THEN
			//Set the category Number
			IF Ldg[Bank].Found = 97 THEN // 97 is weight too small so always set to mixed so it doesn;t get sent to washer..
				myCat = CAT_MIXED_LINEN //Std.MaxCats	- 1
				myPrg = Std.MaxProg	- 1
			ELSE IF (myCat > 0) AND (Bag[StnBag].Cat <> myCat) THEN
				IF (MixCats OR MixProgs) THEN
					//Take the Cat code of bag with most weight
					IF (Bag[StnBag].Wgt > myWgt) THEN
						myCat = Bag[StnBag].Cat
						myPrg = Bag[StnBag].Prg
						myWgt = Bag[StnBag].Wgt
					ENDIF
				ELSE //Different Cats in 1 bag
					myCat = CAT_MIXED_LINEN//Std.MaxCats	- 1
					myPrg = Std.MaxProg - 1
				ENDIF
			ELSE
				myCat = Bag[StnBag].Cat
				myPrg = Bag[StnBag].Prg
				myWgt = Bag[StnBag].Wgt
			ENDIF

			IF (myCus > 0) AND (Bag[StnBag].Cus <> myCus) THEN
				myCus = Std.MaxCust - 1
			ELSE
				myCus = Bag[StnBag].Cus
			ENDIF
		ENDIF

		IF Purge AND (PurgeBagIndex = Std.PurgeBank[myBank].PurgeBagQty) THEN ;Do not minus 1 from purge qty as the indexing is above so will always read 1 more..
			Bag[myBag] 		= Bag[StnBag]
			Bag[StnBag].Mis = 0
			Bag[StnBag].Bid = 0 ; Reset BID

			Bag[myBag].Cat = myCat
			Bag[myBag].Prg = myPrg
			Bag[myBag].Ur2 = 99
			Bag[myBag].Cus	= myCus
			Bag[myBag].Dst 	= USINT(Ldg[myBank].Line)	;Destination
			Bag[myBag].Wgt 	= Std.PurgeBank[myBank].PurgeBatchWieght
			Bag[myBag].Cnt 	= Std.PurgeBank[myBank].PurgeBatchCount

			Bag[myBag].Timestamp = myTimeStamp
			Bag[StnBag].Bid = 0 ; Reset BID
			Bag[StnBag].Dst = 0 					;Reset Destination (Manual)
			Bag[StnBag].Mis = 0
			IF (Ldg[myBank].Found = 98) OR (Ldg[myBank].Found = 97) THEN
	;			D[900 + mySeq] = 3 ;Reverse belt not used.
			ELSE
	;			D[900 + mySeq] = 3
			ENDIF
		ELSE IF NOT Purge AND (Bag[StnBag].Cat <> 98) THEN
			;Copy Station Data to Belt Bag
			Bag[myBag] 		= Bag[StnBag]
			Bag[myBag].Dst 	= USINT(Ldg[myBank].Line)	;Destination
			Bag[myBag].Ur2 = StnBag
			Bag[StnBag].Bid = 0 ; Reset BID
			Bag[StnBag].Dst = 0; USINT(Ldg[myBank].Line) 					;Reset Destination (Manual)
			Bag[StnBag].Mis = 0
			Bag[myBag].Timestamp = myTimeStamp
        	D[900 + mySeq] = 3
		ENDIF
		Alarm[mySeq].Name = almNoAlarm
	ENDIF
ELSE
	Purge = FALSE
	PurgeBagIndex		= 0
	Ldg[myBank].Search  	= 0 ;Clear Search if not on step 2
	myCat = 0
	myPrg = 0
	myCus = 0
	myWgt = 0
ENDIF
ExitStep2:

;;Get batch ID from SQL Server
;IF ((STEP >= 3) AND (STEP <= 4)) THEN
;	IF (Bag[myBag].Mis = 0) THEN
;		_httpRequest;
;	ENDIF
;ELSE
;	HTTP_Comm[myHttp].Status = HTTP_COMM_STATUS_DISABLED
;ENDIF

;Step 3
;Release to Belt Conveyor
TON_10ms(I_PhotoTop,10,LinenDetected,LinenDetectedET)
IF (STEP = 3) THEN
	O_RunBelt = TRUE
	IF LinenDetected OR Test.TransferBelt THEN
		D[900 + mySeq] = 4
	ENDIF
	Alarm[mySeq].Name = almPhotocellNotMade
ENDIF

TON_10ms((STEP = 4),10,RunBelt,Step6ET)
IF (STEP = 4) THEN

	RequestRel.TransferBelt[myBelt] = (Bag[myBag].Cat > 0)
	n = D[900 + Std.StationBankReg + myBank]
	IF EnableRel.TransferBelt[myBelt]  THEN; AND (Bag[myBag].Mis > 0)
		;myTimeStamp = CurrentTimestamp
;		ReportLoading[n].Prg = Bag[290].Prg 			;Program
;		ReportLoading[n].Cat = Bag[290].Cat			;Category
;		ReportLoading[n].Cus = Bag[290].Cus			;Customer
;		ReportLoading[n].Wgt = UINT(WeightValue)		;Weight
;		ReportLoading[n].Cnt = UINT(CountValue)			;Count
;		ReportLoading[n].Stn = n         				;Station
;		ReportLoading[n].Mcn = 0						;Machine
;		ReportLoading[n].Bid = Bag[290].Bid			;Batch ID
;		ReportLoading[n].Mis = Bag[290].Mis
;		ReportLoading[n].TimeStamp = Bag[290].Timestamp
		D[900 + mySeq] = 5
	ENDIF
	IF (Bag[myBag].Cat = 0) THEN
		Alarm[mySeq].Name = almBagDataError
	ELSE IF (Bag[myBag].Mis = 0) THEN
	;	Alarm[mySeq].Name = almBagDataError
	ENDIF

ENDIF

;Step 5 - Run Belt until linen detected for 1 second and Station has emptied
TON_10ms(((STEP = 5) AND I_PhotoTop AND I_InvStatus),50,LinenIsDetected,LinenIsDetectedET)
IF (STEP = 5) THEN
	O_RunBelt = TRUE
	Ldg[myBank].EnableStnRelease = TRUE ;Enable Station to Open bags if they haven't been already
	IF (LinenIsDetected OR Test.TransferBelt)   THEN
		D[900 + mySeq] = 6
	ENDIF
	IF (Bag[myBag].Cat = 0) OR (Bag[myOutBag].Cat > 0) THEN
		Alarm[mySeq].Name = almBagDataError
	ELSE IF NOT Std.HaltSysZone[myZone] THEN
		Alarm[mySeq].Name = almPhotocellNotMade
	ENDIF
ENDIF

;Step 6 - Run Belt until photocells clear for 12 seconds
;TON_10ms((STEP = 6),200,MinimumRun,MinimumRunET)
TON_10ms(((STEP = 6) AND I_InvStatus  AND NOT I_PhotoTop AND NOT Std.HaltSysZone[myZone]),500,BeltClear,BeltClearET)
IF (STEP = 6) THEN
	O_RunBelt = TRUE
	IF (BeltClear AND MinBeltRun AND (Bag[myBag].Cat > 0) AND ((Bag[myOutBag].Cat = 0) OR (Bag[myOutBag].Cat = Std.MaxCats))) THEN
		myBagNumber = Bag[myOutBag].Ur1
		Bag[myOutBag] = Bag[myBag]
		Bag[myOutBag].Ur1 = myBagNumber
		Bag[myBag] = Bag[0]
		D[900 + mySeq] = 7
	ENDIF
	IF NOT Std.HaltSysZone[myZone] THEN
		IF I_PhotoBottom OR I_PhotoTop THEN
			Alarm[mySeq].Name = almPhotocellBlocked
		ELSE IF StationOpen THEN
			Alarm[mySeq].Name = almStationNotClosed
		ELSE IF NOT MinBeltRun THEN
			Alarm[mySeq].Name = almClearingBeltPleaseWait
		ENDIF
	ENDIF
ENDIF

;Step  - Check Stations Are Closed
IF (STEP = 7) THEN
	IF NOT StationOpen AND (Bag[myBag].Cat = 0) THEN
		D[900 + mySeq] = 1
	ENDIF
	Alarm[mySeq].Name = almStationNotClosed
ENDIF

;Note - Unitl the Station has closed the min belt run time won't start
BeltRunTime = (12 + BeltAddTime)
;CTU((O_RunBelt AND Std.Clock1s AND (D[900 + Std.StationBankReg + myBank] = 0) AND NOT Std.EStop),(STEP = 1),BeltRunTime,MinBeltRun,MinBeltRunCV)
BeltRunning = (O_RunBelt OR O_Reverse)
CTU((BeltRunning AND I_InvStatus AND Std.Clock1s AND NOT StationOpen  AND NOT Std.HaltSysZone[myZone]),(STEP = 1),BeltRunTime,MinBeltRun,MinBeltRunCV)

;Slow speed for large load on belt
TON_10ms((NOT I_PhotoLarge AND NOT RunSlow),300,LargeLoadClear,LargeLoadClearET)
IF ((STEP > 2) AND (STEP < 7)) THEN
	IF I_PhotoLarge THEN
		O_SlowBelt = TRUE
	ENDIF
ENDIF

IF (STEP > 0) AND NOT I_InvStatus	THEN
	Alarm[mySeq].Name = almMotorOverload
	Alarm[mySeq].Time = 0
ENDIF

;Alarms
TimerAlarm.IN = NOT PLS AND (Alarm[mySeq].Name > 0)
TimerAlarm.PT = Alarm[mySeq].Time
TimerAlarm FUB TON_10ms()
Alarm[mySeq].On = TimerAlarm.Q
Alarm[mySeq].ET = TimerAlarm.ET

;Outputs
;Inform Station Sequences that the belt has been
Ldg[myBank].BeltHasRun =  (((((D[900 + mySeq] > 3) AND (D[900 + mySeq] < 7)) OR (D[900 + mySeq] >= 10)) AND Ldg[myBank].EnableStnRelease)  OR (D[900 + mySeq] = 1))

Y[11].Y14 = O_RunBelt
//Y[8].Y03 = O_RunBelt AND (STEP < 7) ; Inclined belt... Do not run when reversing.
//Y[8].Y02 = O_Reverse

END_PROGRAM
```

### Program Logical/Sequences/10ms/3_clu_1 (IEC, version 1.00.0) - * Loading unit SLU1

#### 3_slu_1Cyclic.ab
```automation-basic
PROGRAM _CYCLIC
	(* cyclic program *)

;--------------------------------
;Sequence 3 - Loading Unit D[903]
;--------------------------------

;Inputs / Ouputs

;I_BagOutLoadingUnit     = X904
;I_BagSLU1Trip			= X903
;I_BaginLoadingUnit		= X902

EnableRel.TransferBelt[2]	= FALSE
Request.LU[2]                      = FALSE
Request.SP[7]                      = FALSE

I_BagAtBuffer			    = X[3].X03
I_BagFrontPast			  = X[3].X04
I_BagInLoadingUnit		= X[3].X05
I_BagOutCLU1             = X[3].X06

;I_ChuteBlocked			= X[8].X05
;I_CompressorAtTop		= X[5].X13
;I_CompressorAtMid		= X[5].X15
;I_CompressorAtBot		= X[5].X14

O_MoveCompressorUp		= FALSE
O_MoveCompressorDn		= FALSE

I_BagAtSVC1Buffer		= FALSE ;X[12].X11
O_SVC1BufferOpen		= FALSE ;Y[12].Y11

O_OpenBufferStop		= FALSE
O_SteadyCylinders		= FALSE
O_OpenStop	 			= FALSE

RequestRel.LU[2]		= FALSE;
Alarm[3].Name 			= 0
Alarm[3].Bag			= 160
Alarm[3].Beacon			= FALSE
Alarm[3].Extra			= 0
Alarm[3].Time			= 3000

;Setup Sequence
;--------------
STEP = D[903]
;Setup Pulse contact
PLS = (STEP <> LASTSTEP)
LASTSTEP = STEP

IF (STEP = 0) THEN
	;Disabled
ENDIF

;Wait for Empty bag at buffer
SwitchFault = ((STEP = 1) AND (I_BagFrontPast OR I_BagInLoadingUnit))
TON_10ms(NOT SwitchFault,200,LoadingUnitClear,LoadingUnitClearET)
TON_10ms(I_BagAtBuffer,300,BagSettledBuffer,BagSettledBufferET)
IF (STEP = 1) THEN
	IF  BagSettledBuffer AND LoadingUnitClear AND NOT Std.HaltSys THEN
		D[903] = 2
	ENDIF
	IF SwitchFault THEN
		Alarm[3].Name = almSwitchFault
	ELSE
		Alarm[3].Name = almNoAlarm
	ENDIF
ENDIF

IF ((STEP = 2) OR (STEP = 3)) THEN
	Request.SP[7] = TRUE
ENDIF

;Open stops let bag in Loading Unit
IF (STEP = 2) THEN
	O_OpenStop 			= TRUE
	O_OpenBufferStop 	= TRUE
	;Enable.LU[1]		= NOT I_BagFrontPast
	IF I_BagFrontPast THEN
		D[903] = 3
	ENDIF
	Alarm[3].Name = almBagNotArrived
ENDIF

;Wait for bag to settle
TON_10ms(I_BagInLoadingUnit,300,EBagSettled,EBagSettledET)
IF (STEP = 3) THEN
	IF EBagSettled THEN
		D[903] = 4
	ENDIF
	Alarm[3].Name = almBagNotSettled
	;Special for Banbury - SVC1 is also a loading hoist
	;IF SVC1RequestEmpty THEN
	;	Bag[221].Cat 	= 99
	;	D[903] 			= 9
	;ENDIF
ENDIF

;Steady cylinders on from steps 4 - 5
O_SteadyCylinders = ((STEP = 4) OR (STEP = 5))

;Move Steady Cylinders down
TON_10ms((STEP = 4),300,SteadysDown,SteadysDownET)
IF (STEP = 4) THEN
	IF (SteadysDown AND (Bag[160].Cat = 0)) THEN
		D[903] = 5
	ENDIF
	IF (Bag[160].Cat <> 0) THEN
		Alarm[3].Name = almBagDataError
	ELSE
		Alarm[3].Name = almNoAlarm
	ENDIF
ENDIF

;Wait for bag to be loaded
IF (STEP = 5) THEN
;	IF RequestRel.TransferBelt[2] THEN
		EnableRel.TransferBelt[2] = TRUE
;	ENDIF
	IF (Bag[160].Cat > 0) THEN
		D[903] = 6
	ENDIF
	Alarm[3].Name = almNoAlarm ;Transfer belt should alarm
ENDIF

;Allow Steady Cylinders to move up
TON_10ms((STEP = 6),300,SteadysUp,SteadysUpET)
IF (STEP = 6) THEN
	IF SteadysUp AND NOT Enable.LU[2] THEN
			D[903] = 7
	ENDIF
	Alarm[3].Name = almNoAlarm
ENDIF

;Check for space at Buffer
TON_10ms((STEP = 7),300,SteadysUp,SteadysUpET)
IF (STEP = 7) THEN
	IF NOT Std.HaltSys AND SteadysUp AND (Bag[221].Cat = 0) THEN
		Request.LU[2] = TRUE
		IF Enable.LU[2] THEN
			IF (Bag[160].Cat>0) AND (Bag[164].Cat = 0) THEN
							Bag[164] = Bag[160]
							Bag[160] = Bag[0]
			ENDIF
		;	C[34]   = 0
			D[903] 	= 8
			;ELSE
			;Alarm[3].Name = almSwitchFault
		ENDIF
		;ENDIF
	ENDIF
ENDIF

;Open stop - Unitl bag out
IF (STEP = 8) THEN
	O_OpenStop = TRUE
	;IF PLS THEN
	;	C[16] = 0
	;ENDIF
	;IF Line[16].Trip THEN
	IF I_BagOutCLU1  THEN

		D[903] = 1
	ENDIF
	Alarm[3].Name = almBagNotReleased
ENDIF

;Alarms
TimerAlarm.IN = NOT PLS AND (Alarm[3].Name > 0)
TimerAlarm.PT = Alarm[3].Time
TimerAlarm FUB TON_10ms()
Alarm[3].On = TimerAlarm.Q
Alarm[3].ET = TimerAlarm.ET

;Outputs
;-------

Y[3].Y02 = O_OpenBufferStop
Y[3].Y04 = O_SteadyCylinders
Y[3].Y05 = O_OpenStop

;Y[8].Y10 = O_MoveDownTop
;Y[8].Y09 = O_MoveDownBottom
;Y[8].Y15 = O_ElephantsFoot
END_PROGRAM
```

#### 3_slu_1.var
```iecst
VAR RETAIN
	STEP : UINT;
	PLS : BOOL;
	LASTSTEP : UINT;
	EBagSettled : BOOL;
	EBagSettledET : TIME;
	O_OpenStop : BOOL;
	O_SteadyCylinders : BOOL;
	LoadingUnitClear : BOOL;
	LoadingUnitClearET : TIME;
END_VAR
VAR
	CompressCount : UINT;
	O_MoveCompressorUp : BOOL;
	SteadysUpET : TIME;
	SteadysUp : BOOL;
	SteadysDown : BOOL;
	SteadysDownET : TIME;
	I_BagAtBuffer : BOOL;
	O_OpenBufferStop : BOOL;
	I_BagInLoadingUnit : BOOL;
	I_BagFrontPast : BOOL;
	SwitchFault : BOOL;
	TimerAlarm : TON_10ms;
	I_CompressorAtTop : BOOL;
	I_CompressorAtBot : BOOL;
	I_CompressorAtMid : BOOL;
	O_MoveCompressorDn : BOOL;
	BagSettledBuffer : BOOL;
	BagSettledBufferET : TIME;
	I_BagAtSVC1Buffer : BOOL;
	O_SVC1BufferOpen : BOOL;
	I_ChuteBlocked : BOOL;
	CompressorDn : BOOL;
	CompressorDnET : UDINT;
	O_MoveDownTop : BOOL;
	O_MoveDownBottom : BOOL;
	CompressorUp : BOOL;
	CompressorUpET : UDINT;
	O_ElephantsFoot : BOOL;
	I_BagOutCLU1 : BOOL;
END_VAR
```

### Program Logical/Sequences/10ms/4_pn (IEC) - *Ongoing Sequence

#### x_pn.ab
```automation-basic
PROGRAM _CYCLIC

;--------------------------------------
;Sequence 4 - Ongoing To Storage D[900 + mySeq]
;--------------------------------------

;--------------------------------------------------------------------------------
;Revision 1.00 06/11/2009 D.J. First Issue - Automatic Line Allocation with Areas
;--------------------------------------------------------------------------------
mySeq 			= 4
myZone 			= 0
myTransitBag	= 121
myStartStop		= 100

IF (myStartStop >= 100) THEN
	myStartStop = myStartStop + 7600
ENDIF

;Inputs
OnGoingEnable 		= ((D[mySeq] > 0) AND NOT Std.HaltSys)
;I_BagatBuffer[1]	= X715
;I_BagatBuffer[2]	= X716

I_BagatBuffer[1]		= Request.VC[1]
I_BagatBuffer[2]		= X[7].X16
I_BagatBuffer[3]		= FALSE
I_BagatBuffer[4]		= FALSE

O_Reset 		  		= FALSE
O_OpenSelect[1]			= FALSE
O_OpenSelect[2]			= FALSE
O_OpenSelect[3]			= FALSE
O_OpenSelect[4]			= FALSE

O_OpenBuffer[1]			= FALSE
O_OpenBuffer[2]			= FALSE
O_OpenBuffer[3]			= FALSE
O_OpenBuffer[4]			= FALSE

Enable.VC[1]            = FALSE

MaxBuffers 			= 1	;Set Max Buffers to search
MinLine				= 1 	;Set First Storage Line
MaxLine				= 17		;Set Last Storage Line
MaxDepth			= 7    ;Capacity of the longest line - used in search

Alarm[mySeq].Name 		= 0
Alarm[mySeq].Bag		= myTransitBag
Alarm[mySeq].Beacon		= TRUE
Alarm[mySeq].Extra	 	= 0
Alarm[mySeq].Time		= 6000

;Setup Sequence
;--------------
STEP = D[900 + mySeq]
;Setup Pulse contact
PLS = (STEP <> LASTSTEP)
LASTSTEP = STEP

;Step 0 - Disabled
IF (STEP = 0) THEN
	;Disabled
ENDIF

IF SettledBuffer[1] AND (Bag[226].Cat=0) THEN
	Alarm[mySeq].Time		= 6
	Alarm[mySeq].Name       = almBagNotShownOnScreen
ENDIF
IF SettledBuffer[2] AND (Bag[227].Cat=0) THEN
	Alarm[mySeq].Time		= 6
	Alarm[mySeq].Name       = almBagNotShownOnScreen
ENDIF
;Step 1 - Reset Ongoing Points
TON_10ms((STEP = 1),300,ResetPoints,ResetPointsET)
IF (STEP = 1) THEN
	Dest  	= 0
	Buff 	= 0
	O_Reset = TRUE
	IF (ResetPoints AND OnGoingEnable) THEN
		D[900 + mySeq] = 2
	ENDIF
ENDIF

;Bag Settles at each buffer
TON_10ms(I_BagatBuffer[1],300,SettledBuffer[1],SettledBufferET[1])

BufferBagNum[1]	= 120

;BufferBagNum[3]	= myTransitBag

;Step 2 - Search for a valid Bag at one of the buffers
IF (STEP = 2) THEN

	Buff 	= 0
	Dest 	= 0
	BufferDst = 0

	IF OnGoingEnable THEN

		Alarm[mySeq].Name 	= almNoAlarm

		;Search only 1 buffer bag per scan/task
		Buffer = Buffer + 1
		IF Buffer > MaxBuffers THEN
			Buffer = 1
		ENDIF
		;Set Test Value for Monitoring
		IF TestBuffer > 0 THEN
			Buffer = TestBuffer
		ENDIF

		BufferBag		= BufferBagNum[Buffer]
		BufferSettled 	= SettledBuffer[Buffer]
		BufferPrg 		= Bag[BufferBag].Prg
		BufferCat		= Bag[BufferBag].Cat
		BufferCus		= Bag[BufferBag].Cus
		BufferDst 		= Bag[BufferBag].Dst

		IF (BufferSettled AND (BufferCat > 0) AND (BufferPrg > 0) AND (BufferPrg <= Std.MaxProg) AND (OnGoingEnable)) THEN
			IF( (BufferDst>6) OR (BufferDst = 0) )AND Line[23].Clear AND (Line[23].Space>0) THEN
				Dest            = BufferDst
				C[23]           = 0
				D[900 + mySeq] 	= 3
			ENDIF

			;Manual Destination has been set?
			IF (BufferDst > 0) THEN

				n = BufferDst
				IF ((n >= MinLine) AND (n <= MaxLine) AND (Line[n].Space > 0) AND Line[n].Clear) THEN
					Dest 	= n
					Buff 	= Buffer
					D[900 + mySeq] 	= 3
				ELSE
					Alarm[mySeq].Name 	= almDestinationNotValid
					Alarm[mySeq].Bag	= BufferBag
				ENDIF

			ELSE IF Std.AutoLineAllocation THEN ;/BufferDst > 0

				;Search Each Storage Area
				AreaChoice[1] = D[3000 + BufferPrg]
				AreaChoice[2] = D[3100 + BufferPrg]
				AreaChoice[3] = D[3200 + BufferPrg]
				AreaChoice[4] = D[3300 + BufferPrg]

				LOOP Area = 1 TO 4 DO

					AreaStartLine 	= D[250 + AreaChoice[Area]]
					AreaEndLine 	= D[270 + AreaChoice[Area]]
					AreaValid		= ((AreaStartLine > 0) AND (AreaEndLine > 0) AND (AreaEndLine >= AreaStartLine))
					IF AreaValid THEN

						;Search for a line with the same program
						;---------------------------------------
						LOOP myLine = AreaStartLine TO AreaEndLine DO
							myLineValid = ((myLine >= MinLine) AND (myLine <= MaxLine))
							myLineUsed	= (D[myStartStop + myLine] > 0) ;Start / Stop On
							IF myLineValid AND myLineUsed THEN
								n 			= myLine
								SearchBag 	= (Line[n].LastBag - Line[n].Space)
								IF ((SearchBag >= Line[n].FirstBag) AND (Bag[SearchBag].Prg = BufferPrg) AND (Line[n].Space > 0) AND Line[n].Clear) THEN
									;Found line with a matching program
									Dest 	= n
								ENDIF ;/SearchBag
							ENDIF ;/myLineValid
							EXITIF (Dest <> 0)
						ENDLOOP ;/myLine loop

						;Search for an empty line
						;------------------------
						IF (Dest = 0) THEN
							LOOP myLine = AreaStartLine TO AreaEndLine DO
								myLineValid = ((myLine >= MinLine) AND (myLine <= MaxLine))
								myLineUsed	= (D[myStartStop + myLine] > 0) ;Start / Stop On
								IF myLineValid AND myLineUsed THEN
									n 			= myLine
									SearchBag 	= (Line[n].FirstBag)
									IF ((Bag[SearchBag].Prg = 0) AND (Line[n].Space > 0) AND Line[n].Clear) THEN
										;Found line with a matching program
										Dest 	= n
									ENDIF ;/SearchBag
								ENDIF ;/myLineValid
							EXITIF (Dest <> 0)
							ENDLOOP ;/myLine loop
						ENDIF ;/Dest = 0

						;Search for a line that already contains a bag with the same program starting at the back
						;----------------------------------------------------------------------------------------
						IF (Dest = 0) THEN
							LOOP myDepth = (MaxDepth - 2) DOWNTO 0 DO ;Don't search the last bag as the line would already be full!!
								LOOP myLine = AreaStartLine TO AreaEndLine DO
									myLineValid = ((myLine >= MinLine) AND (myLine <= MaxLine))
									myLineUsed	= (D[myStartStop + myLine] > 0) ;Start / Stop On
									IF myLineValid AND myLineUsed THEN
										n 			= myLine
										SearchBag 	= (Line[n].FirstBag + myDepth)
										IF ((Bag[SearchBag].Prg = BufferPrg) AND (Line[n].Space > 0) AND Line[n].Clear) THEN
											;Found line with a matching program
											FoundDepth 	= myDepth
											Dest 		= n
										ENDIF ;/SearchBag
									ENDIF ;/myLineValid
									EXITIF (Dest <> 0)
								ENDLOOP ;/myLine loop
								EXITIF (Dest <> 0)
							ENDLOOP ;/myDepgh
						ENDIF ;/Dest = 0

						;Search for line with the most space
						;-----------------------------------
						IF (Dest = 0) THEN
							mySpace = 0
							myFound	= 0
							LOOP myLine = AreaStartLine TO AreaEndLine DO
								myLineValid = ((myLine >= MinLine) AND (myLine <= MaxLine))
								myLineUsed	= (D[myStartStop + myLine] > 0) ;Start / Stop On
								IF myLineValid AND myLineUsed THEN
									n 			= myLine
									SearchBag 	= (Line[n].LastBag)
									IF ((Bag[SearchBag].Prg = 0) AND (Line[n].Space > mySpace) AND Line[n].Clear) THEN
										;Found line with a matching program
										myFound	= n
										mySpace = Line[n].Space
									ENDIF ;/SearchBag
								ENDIF ;/myLineValid
							ENDLOOP ;/myLine loop

							IF (myFound > 0) THEN
								Dest 	= myFound
							ENDIF

						ENDIF ;/Dest = 0

					ENDIF ;/Area Valid
					EXITIF (Dest <> 0)
				ENDLOOP ;/Area Loop

			ENDIF ;/BufferDst > 0

			;Destination line found!!
			IF (Dest <> 0) THEN
				Buff = Buffer
				IF (Bag[myTransitBag].Cat = 0) AND (Bag[BufferBagNum[Buff]].Cat > 0) THEN ;Bag in Transit
					Bag[BufferBagNum[Buff]].Dst = USINT(Dest)
					Bag[myTransitBag]	= Bag[BufferBagNum[Buff]]
					Bag[BufferBagNum[Buff]]	 	= Bag[0]
					IF(Dest < 7) THEN
						C[Dest] = 0
					ENDIF
					D[900 + mySeq] 	= 3 ; Open buffer
				ENDIF
			ELSE
				;Storage full!!
				;Do Nothing? Alarm?
				;Other Area?
			ENDIF

		ENDIF ;/BagSettled

		;Buffer Alarms
		IF (BufferPrg > 0) AND NOT BufferSettled THEN
		;	Alarm[mySeq].Name 	= almBagNotAtProx
		;	Alarm[mySeq].Bag	= BufferBag
		ELSE IF (BufferPrg = 0) AND BufferSettled THEN
			Alarm[mySeq].Name 	= almBagNotShownOnScreen
			Alarm[mySeq].Bag	= BufferBag
		ENDIF
	ENDIF
ENDIF

;Clear Line Selections
LOOP n = 1 TO Std.MaxLines DO
	LineSelect[n] = FALSE
ENDLOOP

;Step 3 - Select line / open buffer stop
IF (STEP = 3) THEN
	IF (Bag[myTransitBag].Cat = 0) AND (Bag[120].Cat > 0) THEN ;Bag in Transit
			;Bag[BufferBagNum[Buff]].Dst = USINT(Dest)
			Bag[myTransitBag]	= Bag[120]
			Bag[120]	 	= Bag[0]
			C[23] = 0

	ENDIF
	Enable.VC[1]       = TRUE
	LineSelect[Dest]   = TRUE
	O_OpenBuffer[Buff] = TRUE
	IF ((Dest> 6) OR (Dest = 0)) AND Line[23].Trip THEN
		IF (Bag[134].Cat = 0) AND (Bag[121].Cat > 0) THEN
			Bag[134] = Bag[121]
			Bag[121] = Bag[0]
		ENDIF
		D[900 + mySeq] 				= 1
	ENDIF
	;Bag arrived on selected line
	IF Line[Dest].Trip THEN
		D32[498] 					= Bag[myTransitBag].Cus	;Set Customer for Customer FIFO
		Bag[myTransitBag].Dst 		= 0 		    ;Clear Destination
		Bag[Line[Dest].LastBag] 	= Bag[myTransitBag]
		Bag[myTransitBag] 			= Bag[0]
		D[900 + mySeq] 				= 1
	ENDIF
	Alarm[mySeq].Time		= 6000
	Alarm[mySeq].Name = almBagNotArrived
ENDIF

;Alarms
TimerAlarm.IN = NOT PLS AND (Alarm[mySeq].Name > 0) AND (AlarmOld = Alarm[mySeq].Name)
TimerAlarm.PT = Alarm[mySeq].Time
TimerAlarm FUB TON_10ms()
Alarm[mySeq].On = TimerAlarm.Q
Alarm[mySeq].ET = TimerAlarm.ET

AlarmOld = Alarm[mySeq].Name ;Need to ensure alarm changes as may be multiple alarms on step 2

;Y[6].Y09 = O_OpenBuffer[1]

;Outputs
Y[4].Y09 = O_Reset OR (Dest > 6)
Y[4].Y01 = LineSelect[1]
Y[4].Y02 = LineSelect[2]
Y[4].Y03 = LineSelect[3]
Y[4].Y04 = LineSelect[4]
Y[4].Y05 = LineSelect[5]
Y[4].Y06 = LineSelect[6]

END_PROGRAM
```

### Program Logical/Sequences/10ms/5_pf (IEC) - *Offgoing Sequence

#### pf1.var
```iecst
VAR RETAIN
	LASTSTEP : UINT;
	SelectedBuffer : USINT;
	Destination : UINT;
	FoundLine : UINT;
END_VAR
VAR
	x : UINT;
	Line14_Valid : BOOL;
	LongestLine : UINT;
	O_Select : ARRAY[0..22] OF BOOL;
	LongestSTime : UINT;
	LineInList : ARRAY[0..98] OF BOOL;
	mySeq : UINT;
	RecircSpaces : UINT;
	O_Reset3way : BOOL;
	r : UINT;
	myRelLine : UINT;
	SettleTime : UINT;
	TransitBag : UINT;
	RecircValid : BOOL;
	TimerAlarm : TON_10ms;
	SDC6_Valid : BOOL;
	SDC5_Valid : BOOL;
	SDC7_Valid : BOOL;
	TestAtStop : BOOL;
	STEP : UINT;
	SDC3_Valid : BOOL;
	SearchDest : UINT;
	SDC4_Valid : BOOL;
	I_InclineBufferStopOpen : BOOL;
	ResetPointsET : TIME;
	ResetPoints : BOOL;
	OffGoingEnable : BOOL;
	SDC1_Valid : BOOL;
	SDC2_Valid : BOOL;
	PLS : BOOL;
	O_SDCBufferOpen : ARRAY[0..4] OF BOOL;
	O_Reset : BOOL;
	MaxLine : UINT;
	n : UINT;
	MinLine : UINT;
	BufferBag : ARRAY[0..9] OF UINT;
	LineSelect : ARRAY[0..30] OF BOOL;
	MaxBuffers : UINT;
	I_SDCBagAtBuffer : ARRAY[0..4] OF BOOL;
	I_BagAtIncline : BOOL;
	IncSettle : BOOL;
	LineSettle : ARRAY[0..30] OF BOOL;
	BestTime : UINT;
	BufferClear : ARRAY[0..9] OF BOOL;
	AlarmBagNotProx : BOOL;
	I_BagAtStop : ARRAY[0..30] OF BOOL;
	BagSettledTime : ARRAY[0..30] OF UINT;
	myZone : UINT;
	I_BagAtWeighbeam : BOOL;
	I_BagOutOfBeam : BOOL;
	BagAtBeam : BOOL;
	OpenSpeedReducor : BOOL;
	OpenSpeedReducorET : UDINT;
END_VAR
```

#### pf1.ab
```automation-basic
PROGRAM _CYCLIC

;----------------------------------------
;Sequence 5 - SPF1 Offgoing Points D[900+mySeq]
;----------------------------------------

;Inputs
;------
mySeq			= 5
myRelLine 		= 0
TransitBag 		= 155
myZone			= 0

OffGoingEnable 		= ((D[mySeq] > 0) AND NOT Std.HaltSysZone[myZone])

I_SDCBagAtBuffer[1] = FALSE ;Bag In Discharger
I_SDCBagAtBuffer[2] = FALSE ;Use for single bag buffer
I_SDCBagAtBuffer[3] = FALSE ;X[6].X13 ;Use for single bag buffer
I_SDCBagAtBuffer[4] = FALSE ;X[6].X13 ;Use for single bag buffer

O_SDCBufferOpen[1]  = FALSE ;Use for single bag buffer
O_SDCBufferOpen[2]  = FALSE ;Use for single bag buffer
O_SDCBufferOpen[3]  = FALSE ;Y[6].Y16 ;Use for single bag buffer
O_SDCBufferOpen[4]  = FALSE ;Y[6].Y16 ;Use for single bag buffer

I_BagAtStop[1]	 	= X[5].X01 OR TestAtStop
I_BagAtStop[2] 		= X[5].X02 OR TestAtStop
I_BagAtStop[3] 		= X[5].X03 OR TestAtStop
I_BagAtStop[4] 		= X[5].X04 OR TestAtStop
I_BagAtStop[5]	 	= X[5].X05 OR TestAtStop
I_BagAtStop[6] 		= X[5].X06 OR TestAtStop

O_Reset 			= FALSE

;Buffer line configuration
;-------------------------
MaxBuffers			= 1
MinLine				= 1
MaxLine				= 6

;BufferBag[1]		= 251 ;Last buffer bag number
;BufferBag[2]		= 373;Last buffer bag number
;BufferBag[3]		= 383 ;Last buffer bag number CDC3
;BufferBag[4]		= 192 ;Last buffer bag number CDC4
;BufferBag[5]		= 155 ;Last buffer bag number CDC 5
;BufferBag[6]		= 658 ;Last buffer bag number
;BufferBag[7]		= 664 ;Last buffer bag number
;RecircSpaces  		=(Line[20].Space + Line[24].Space + (Bag[190].Cat = 0) - DestCountSystem[30])

;BufferClear[1] 		= ((D[6]> 0) AND (Line[31].SpaceBIT > 0) )
;BufferClear[2]		= ((Bag[Line[22].LastBag].Cat = 0) AND  (Line[22].SpaceBIT >= 1)); Empty bag buffer before CDC2
;BufferClear[3]		= ((Bag[Line[23].LastBag].Cat = 0) AND  (Line[23].SpaceBIT >= 1))
;BufferClear[4]		= (Bag[BufferBag[4]].Cat = 0) AND (RecircSpaces > 0) ;Recirc Valid
;BufferClear[5]		= ((Bag[BufferBag[5]].Cat = 0) AND (D[10] > 0) AND Request.DC[5] AND (Line[25].SpaceBIT >= 1))
;;BufferClear[6]		= (D[9] > 0) AND (Bag[BufferBag[6]].Cat = 0)
;BufferClear[7]		= (D[10] > 0) AND (Bag[BufferBag[7]].Cat = 0)
Uld[1].SDCReady 	= ((D[21] > 0)AND (Line[11].SpaceBIT > 0))
Uld[2].SDCReady 	= ((D[22] > 0)AND (Line[12].SpaceBIT > 0))

Uld[3].SDCReady		= ((D[23] > 0)AND (Line[13].SpaceBIT > 0))
Uld[4].SDCReady 	= FALSE
;Uld[5].SDCReady 	= BufferClear[5]

Alarm[mySeq].Name 		= 0
Alarm[mySeq].Bag		= TransitBag
Alarm[mySeq].Beacon		= TRUE
Alarm[mySeq].Extra		= 0
Alarm[mySeq].Time		= 4500

;Setup Sequence
;--------------
STEP = D[900 + mySeq]
;Setup Pulse contact
PLS = (STEP <> LASTSTEP)
LASTSTEP = STEP

;Sequence Steps
;--------------
IF (STEP = 0) THEN
	;Disabled
ENDIF

;Step 1 - Reset Points
TON_10ms((STEP = 1),300,ResetPoints,ResetPointsET)
IF (STEP = 1) THEN
	O_Reset 	= NOT ResetPoints
	FoundLine 	= 0
	Destination = 0
	IF (ResetPoints AND OffGoingEnable) THEN
		D[900+mySeq] = 2
	ENDIF
ENDIF

;Bags on storage line timers
R_TRIG(Std.Clock100ms,IncSettle)
AlarmBagNotProx 	= FALSE
AlarmBagNotProxLine = 0

LOOP n = MinLine TO MaxLine DO

	LineSettle[n]  = (I_BagAtStop[n] AND (Bag[Line[n].FirstBag].Cat > 0))
	IF IncSettle AND LineSettle[n] AND (BagSettledTime[n] < $FFFF) THEN
		BagSettledTime[n] = BagSettledTime[n] + 1
	ELSE IF NOT LineSettle[n] THEN
		BagSettledTime[n] = 0
		;If Bag has destiantion and not at stop then alarm
		IF (Bag[Line[n].FirstBag].Dst > 0) THEN
			Alarm[mySeq].Name	= almBagNotAtProx
			Alarm[mySeq].Bag	= Line[n].FirstBag
			Alarm[mySeq].Extra 	= n
		ENDIF
	ENDIF
	IF (I_BagAtStop[n] AND (Bag[Line[n].FirstBag].Cat = 0)) THEN
		;Alarm[mySeq].Name	= almSwitchFault
		;	Alarm[mySeq].Bag	= Line[n].FirstBag
		;	Alarm[mySeq].Extra 	= n
	ENDIF
		LongestSTime = 0
		LongestTime[n] = 0
ENDLOOP

LOOP n = MinLine TO MaxLine DO
	LineInList[n]  = FALSE
ENDLOOP

LOOP n = MinLine TO MaxLine DO
	LongestLine = 0
	LongestSTime = 0
	LOOP x = MinLine TO MaxLine DO
		IF (BagSettledTime[x] > LongestSTime) AND NOT LineInList[x] THEN ;(BagSettledTime[x] > BagSettledTime[n]) AND
			LongestSTime = BagSettledTime[x]
			LongestLine = x
		ENDIF
	ENDLOOP
	LineInList[LongestLine] = TRUE
	LongestTime[n] = LongestLine
ENDLOOP

;Buffer trip not correct alarms
LOOP n = 1 TO MaxBuffers DO
	IF (STEP = 2) AND  NOT Uld[n].SDCReady THEN
		;Alarm[mySeq].Name 	= almSwitchFault - Not direct to buffers
		;Alarm[mySeq].Bag	= BufferBag[n]
	ENDIF
ENDLOOP

;Search for the bag with a valid destination that has been waiting the longest
IF STEP = 2 THEN

	FoundLine 	= 0
	Destination = 0
	BestTime 	= 0
	SettleTime = 30 ;3 seconds

	LOOP n = MinLine TO MaxLine DO
		IF ((BagSettledTime[n] > SettleTime) AND (BagSettledTime[n] > BestTime)) THEN
			SearchDest = Bag[Line[n].FirstBag].Dst

			SDC1_Valid  = (SearchDest = 11) AND Uld[1].SDCReady
			SDC2_Valid 	= (SearchDest = 12) AND Uld[2].SDCReady
			SDC3_Valid 	= (SearchDest = 13) AND Uld[3].SDCReady
;			SDC4_Valid 	= (SearchDest = 34) AND Uld[4].SDCReady
;			SDC5_Valid 	= ((SearchDest = 35) AND Uld[5].SDCReady)
            ;SDC6_Valid 	= ((SearchDest = 36) AND Uld[6].SDCReady)
			;SDC7_Valid 	= ((SearchDest = 37) AND Uld[7].SDCReady)
			;RecircValid = ((SearchDest = 30) AND Line[20].Clear AND (Bag[Line[20].LastBag].Cat = 0))
			IF SDC1_Valid OR SDC2_Valid or SDC3_Valid THEN
				FoundLine 	= n
				Destination = SearchDest
				BestTime 	= BagSettledTime[n]
			ENDIF
		ENDIF
	ENDLOOP

	IF ((FoundLine > 0) AND (Destination > 0) AND OffGoingEnable AND (Bag[TransitBag].Cat = 0)) THEN
		IF  (Bag[TransitBag] .Cat = 0) AND Line[21].Clear AND NOT X[9].X01 AND NOT Y[5].Y11 AND (Bag[165].Cat = 0) THEN ;AND ((Request.DC[1] AND NOT X[3].X10) OR  (Request.DC[2] AND NOT X[3].X13)) THEN

			C[21] = 0
			D[900 + mySeq] = 3
		ENDIF
	ENDIF
ENDIF

;Step 3 - Select Line / Open Stop, Until Bag at correct destination
;Clear Line Selections
LOOP n = MinLine TO MaxLine DO
	LineSelect[n] = FALSE
ENDLOOP

TON_10ms((STEP = 3) AND BagAtBeam,300,OpenSpeedReducor,OpenSpeedReducorET)
IF (STEP = 3) THEN
	LineSelect[FoundLine] = TRUE
	IF (Destination >= 11) AND (Destination <= 13) THEN
		Uld[Destination - 10].DischargerStartLine = FoundLine ;Unloading Program
	ENDIF
	IF (Bag[TransitBag] .Cat = 0) AND (Bag[Line[FoundLine].FirstBag].Cat > 0)THEN
		IF PLS THEN
			Bag[TransitBag]  = Bag[Line[FoundLine].FirstBag]
			Bag[Line[FoundLine].FirstBag] 	= Bag[0]
		ENDIF
	ENDIF
	IF (((Destination = 11) OR  (Destination = 12)OR  (Destination = 13))AND Line[21].Trip) THEN
		Bag[165] = Bag[TransitBag]
		Bag[TransitBag] = Bag[0]
		D[900 + mySeq] = 1
	ENDIF

	Alarm[mySeq].Name	= almBagNotReleased
ENDIF

;Alarms
TimerAlarm.IN = NOT PLS AND (Alarm[mySeq].Name > 0)
TimerAlarm.PT = Alarm[mySeq].Time
TimerAlarm FUB TON_10ms()
Alarm[mySeq].On = TimerAlarm.Q
Alarm[mySeq].ET = TimerAlarm.ET

;Outputs
;-------

;Y[5].Y07 = O_Reset

Y[5].Y01 = LineSelect[1]
Y[5].Y02 = LineSelect[2]
Y[5].Y03 = LineSelect[3]
Y[5].Y04 = LineSelect[4]
Y[5].Y05 = LineSelect[5]
Y[5].Y06 = LineSelect[6]
Y[5].Y07 = LineSelect[7] OR O_Reset

;Y[12].Y06 = OpenSpeedReducor

END_PROGRAM
```

### Program Logical/Sequences/10ms/6_sdc1 (IEC, version 1.00.0) - * SDC1 Machine 1 BIN/BCD

#### 6_sdc1Cyclic.ab
```automation-basic
PROGRAM _CYCLIC
	(* cyclic program *)

;Sequence 6 - Discharger 1 D[906]

;-----------------------------------------
;Revision 1.00 19/12/2005 D.J. First Issue
;-----------------------------------------

DischargerEnable 		= ((D[11] > 0) AND NOT Std.HaltSys)

I_OpenBag				= (CAN[1].DropLoad );	AND CAN[1].ReadyToLoad)
I_LoadDropped			= CAN[1].LoadDropped
I_BagAtBuffer			= X[6].X05
I_BagAtDischarger		= X[6].X06

I_BagEmpty			  	= TRUE

I_BagAtEmptyBuffer		= FALSE ;X[11].X07
O_EmptyBagBufferOpen	= FALSE ;Y[11].Y07
Request.SDC1Drop        = FALSE
Request.DCEmptyRelease[1] = FALSE
O_BagReady				= FALSE
O_OpenBuffer 			= FALSE
O_Steadys				= FALSE
O_Closer				= FALSE
O_OpenBag				= FALSE
O_OpenStop				= FALSE

Request.DC[1]			= FALSE
Request.SDC1Drop        = FALSE

;Alarm
Alarm[6].Name 			= almNoAlarm ;Clear sequence alarm name
Alarm[6].Bag 			= 50
Alarm[6].Beacon			= TRUE
Alarm[6].Extra			= 0
Alarm[6].Time			= 3000

;Setup Sequence
STEP = D[906]
;Setup Pulse contact
PLS = (STEP <> LASTSTEP)
LASTSTEP = STEP

;Step 0 - Disabled
IF (STEP = 0) THEN
	;Disabled
ENDIF

;Check Status - Bag settled at buffer, no bag at discharger, bag at buffer on screen and no bag at discharger on the screen
TON_10ms(I_BagAtBuffer,300,SettledAtBuffer,SettledAtBufferET)
IF (STEP = 1) THEN
	Request.DC[1] = DischargerEnable
	IF (NOT I_BagAtDischarger AND  (Bag[50].Cat = 0) AND (Bag[51].Cat > 0)AND NOT Std.HaltSys AND DischargerEnable AND SettledAtBuffer) THEN
		;Request.DC[1] = TRUE
		D[906] = 2
	ENDIF
	IF I_BagAtDischarger THEN
		;D[906] = 2
	ENDIF
	IF (Bag[50].Cat > 0) THEN
		Alarm[6].Name = almBagDataError
	ELSE IF I_BagAtDischarger THEN
		Alarm[6].Name = almSwitchFault
	ELSE IF (Bag[51].Cat > 0) AND NOT I_BagAtBuffer THEN
		Alarm[6].Name 	= almBagNotAtProx
		Alarm[6].Bag	= 51
	ELSE IF (Bag[51].Cat = 0) AND I_BagAtBuffer AND DischargerEnable  THEN
		Alarm[6].Name 	= almBagNotShownOnScreen
		Alarm[6].Bag	= 51
	ENDIF
ENDIF

;Wait for bag in discharger
IF (STEP = 2) THEN
	O_OpenBuffer 	= TRUE
	IF I_BagAtDischarger THEN
		D[906] = 3
	ENDIF
	Alarm[6].Name = almBagNotArrived
ENDIF

;Let bag settle in discharger
TON_10ms(((STEP = 3) AND I_BagAtDischarger),1000,SettledAtDischarger,SettledAtDischargerET)
IF (STEP = 3) THEN
	IF PLS  AND (Bag[50].Cat = 0) AND (Bag[51].Cat > 0) THEN
		Bag[50] = Bag[51]
		Bag[51] = Bag[0]
	ENDIF
	IF SettledAtDischarger THEN
		D[906] = 4
	ENDIF
	;IF ((Bag[280].Cat > 0) AND (Bag[280].Dst = 23)) THEN
	;	D[906] = 11
	;ENDIF
	Alarm[6].Name = almBagNotSettled
ENDIF

IF (D[981] = 0) AND (STEP = 6) THEN
	IF (Bag[51].Cat>0) AND (Bag[50].Cat>0) AND (Bag[51].Cat = Bag[50].Cat) THEN
		D[981] = 2
	ELSE
		D[981] = 1
	ENDIF
ENDIF

IF (D[981] = 1) AND( (STEP = 6) OR (STEP = 7) OR (STEP = 8)) THEN
	CAN[1].LoadFinished = TRUE
ELSE
	CAN[1].LoadFinished = FALSE
ENDIF

;Allow steadys to move down
TON_10ms((STEP = 4),400,SteadysDown,SteadysDownET)
IF (STEP = 4) THEN
	IF SteadysDown AND ((Bag[51].Cat>0) OR (D[981]=1)) THEN
		D[906] = 5
	ENDIF
	IF (Bag[50].Cat = Std.MaxCats) THEN
		D[906] = 8
	ENDIF
ENDIF

;Steady cylinders on from steps 4 - 9
O_Steadys = ((STEP >= 4) AND (STEP <= 9))

;Bag opener on from step 5 - 8
O_OpenBag = ((STEP >= 6) AND (STEP <= 8))

CodeStep  = ((STEP >= 4) AND (STEP <= 5))

;Wash Codes
;Wash Codes
IF CodeStep THEN
	Weight = Bag[50].Wgt
	;round up weight to give to wash machine
	Remainder = SINT(Weight MOD 10)
	IF (Remainder > 4) THEN
		WgtRound = (Weight + 10)
	ELSE
		WgtRound = Weight
	ENDIF

	CAN[1].Category = Bag[50].Cat
	CAN[1].Customer = Bag[50].Cus
	CAN[1].Weight   = (WgtRound / 10)
ELSE
	CAN[1].Category = 0
	CAN[1].Customer = 0
	CAN[1].Weight   = 0
ENDIF

;Bag Ready to Washing Machine
IF (STEP = 5) THEN
	O_BagReady = (Bag[50].Cat > 0)
	IF I_OpenBag THEN
		D[906] = 6
	ENDIF
	IF (Bag[50].Cat = 0) THEN
		Alarm[6].Time = 1
		Alarm[6].Name = almBagNotShownOnScreen
	ENDIF
	ELSE
	O_BagReady = FALSE
ENDIF

;Set LoadDropped to False
IF (STEP <> 6) THEN
	LoadDropped = FALSE
ENDIF

;Open Bag Until LoadDropped recieved and has been open for 6 seconds
TON_10ms((STEP = 6),600,MinOpen,MinOpenET) ;ET means Elapsed Time
IF (STEP = 6) THEN

	IF I_LoadDropped OR TestDischarger THEN
	;IF I_BagEmpty THEN
		LoadDropped = TRUE
	ENDIF

	IF (LoadDropped AND MinOpen) THEN
		;Write Report
		;------------
		IF (ReportUnloading[1].Cat = 0) THEN
			ReportUnloading[1].Cat = UINT(Bag[50].Cat)	;Category
			ReportUnloading[1].Cus = Bag[50].Cus		;Customer
			ReportUnloading[1].Wgt = Bag[50].Wgt		;Weight
			ReportUnloading[1].Cnt = 0					;Count
			ReportUnloading[1].Stn = 0					;Station
			ReportUnloading[1].Mcn = 1					;Machine
		ENDIF
	ENDIF
	IF (LoadDropped AND MinOpen) THEN
		D[906] = 7
	ENDIF
	Alarm[6].Name = almLoadNotDropped
ENDIF

;Change display to empty bag
IF (STEP = 7) THEN

	IF ((NOT  I_OpenBag AND NOT I_LoadDropped AND I_BagEmpty) OR TestDrop) THEN
		Bag[50].Prg 	= Std.MaxProg
		Bag[50].Cat 	= Std.MaxCats
		Bag[50].Cus 	= Std.MaxCust
		D[906] 			= 8
	ENDIF
	Alarm[6].Name = almSwitchFault
ENDIF

;Close bag
TON_10ms((STEP = 8),700,CloserDown,CloserDownET)
IF (STEP = 8) THEN
	O_Closer = TRUE
	IF CloserDown THEN
		D[906] = 9
	ENDIF
;	CAN[1].LoadFinished= TRUE
	ELSE
;	CAN[1].LoadFinished = FALSE
ENDIF

;Allow closer to go back up
TON_10ms((STEP = 9),700,CloserUp,CloserUpET)
IF (STEP = 9) THEN
	IF PLS THEN
		IF (D[981]>0) THEN
			D[981] = (D[981]-1)
		ENDIF
	ENDIF
	IF CloserUp THEN
		D[906] = 10
	ENDIF
ENDIF

;Allow steadys to go up
TON_10ms((STEP = 10),400,SteadyUp,SteadyUpET)
IF (STEP = 10) THEN
	IF SteadyUp  THEN
		D[906] = 11
	ENDIF
ENDIF

;Check for space on empty bag buffer
IF (STEP = 11) THEN
	;Request.DCEmptyRelease[1] = TRUE
	IF Line[34].Clear THEN
		C[34]  = 0
		D[906] = 12
	ENDIF
ENDIF

;Open buffer stop - unitl bag out
IF (STEP = 12) THEN
	O_OpenStop = TRUE
	;IF PLS THEN
	;	C[25] = 0
	;ENDIF
	Bag[50].Cat = 0
	Bag[50].Cus = 0
	Bag[50].Wgt = 0
	IF Line[34].Trip THEN
		D[906] = 1
	ENDIF
	Alarm[6].Name = almBagNotReleased
ENDIF

;Alarms
TimerAlarm.IN 	= NOT PLS AND (Alarm[6].Name > 0)
TimerAlarm.PT 	= Alarm[6].Time
TimerAlarm FUB TON_10ms()
Alarm[6].On 	= TimerAlarm.Q
Alarm[6].ET 	= TimerAlarm.ET

;Outputs
CAN[1].BagReady = O_BagReady
Y[6].Y01 			= O_OpenBuffer
Y[6].Y02 			= O_Steadys
Y[6].Y03 			= O_OpenBag
Y[6].Y04 			= O_Closer
Y[6].Y05 			= O_OpenStop
END_PROGRAM
```

#### 6_sdc1.var
```iecst
VAR RETAIN
	STEP : UINT;
	PLS : BOOL;
	LASTSTEP : UINT;
	SteadyUp : BOOL;
	CloserUpET : TIME;
	SteadysDown : BOOL;
	SteadysDownET : TIME;
	LoadDropped : BOOL;
	SteadyUpET : TIME;
	CloserDownET : TIME;
	SettledAtDischargerET : TIME;
	MinOpenET : TIME;
	SettledAtDischarger : BOOL;
	CloserDown : BOOL;
	MinOpen : BOOL;
	CloserUp : BOOL;
	SettledAtBuffer : BOOL;
	SettledAtBufferET : TIME;
	I_BagAtBuffer : BOOL;
	O_OpenStop : BOOL;
	O_OpenBag : BOOL;
	O_Steadys : BOOL;
	O_OpenBuffer : BOOL;
	O_Closer : BOOL;
	I_BagAtDischarger : BOOL;
	I_OpenBag : BOOL;
	I_LoadDropped : BOOL;
	TestDrop : BOOL;
END_VAR
VAR
	DischargerEnable : BOOL;
	TestDischarger : BOOL;
	I_BagEmpty : BOOL;
	O_BagReady : BOOL;
	I_BagReleased : BOOL;
	O_EmptyBagBufferOpen : BOOL;
	I_BagAtEmptyBuffer : BOOL;
	TimerAlarm : TON_10ms;
	CodeStep : BOOL;
	BCD_BIN_CAT : BCD_BIN_OUTPUT;
	BCD_BIN_CUS : BCD_BIN_OUTPUT;
	BCD_BIN_WGT : BCD_BIN_OUTPUT;
	Remainder : UINT;
	WgtRound : UINT;
	Weight : UINT;
END_VAR
```

### Program Logical/Sequences/10ms/7_sdc2 (IEC) - * SDC2 Machine 2 CAN

#### 7_sdc2.var
```iecst
VAR RETAIN
	STEP : UINT;
	PLS : BOOL;
	LASTSTEP : UINT;
	SteadyUp : BOOL;
	CloserUpET : TIME;
	SteadysDown : BOOL;
	SteadysDownET : TIME;
	LoadDropped : BOOL;
	SteadyUpET : TIME;
	CloserDownET : TIME;
	SettledAtDischargerET : TIME;
	MinOpenET : TIME;
	SettledAtDischarger : BOOL;
	CloserDown : BOOL;
	MinOpen : BOOL;
	CloserUp : BOOL;
	SettledAtBuffer : BOOL;
	SettledAtBufferET : TIME;
	I_BagAtBuffer : BOOL;
	O_OpenStop : BOOL;
	O_OpenBag : BOOL;
	O_Steadys : BOOL;
	O_OpenBuffer : BOOL;
	O_Closer : BOOL;
	I_BagAtDischarger : BOOL;
	I_OpenBag : BOOL;
	I_LoadDropped : BOOL;
	TestDrop : BOOL;
END_VAR
VAR
	DischargerEnable : BOOL;
	TestDischarger : BOOL;
	I_BagEmpty : BOOL;
	O_BagReady : BOOL;
	WgtRound : UINT;
	TimerAlarm : TON_10ms;
	I_BagReleased : BOOL;
	O_EmptyBagBufferOpen : BOOL;
	I_BagAtEmptyBuffer : BOOL;
	Remainder : UINT;
	CodeStep : BOOL;
	I_DischargerBagEmpty : BOOL;
	BagEmpty : BOOL;
	BagEmptyET : TIME;
	BCD_BIN_CAT : BCD_BIN_OUTPUT;
	BCD_BIN_CUS : BCD_BIN_OUTPUT;
	BCD_BIN_WGT : BCD_BIN_OUTPUT;
	TestDropped : BOOL;
	TestBuffer : BOOL;
	TestAtDisch : BOOL;
	Weight : UINT;
	KEV : BOOL;
END_VAR
```

#### 7_sdc2Cyclic.ab
```automation-basic
PROGRAM _CYCLIC
	(* cyclic program *)

;Sequence 7 - Discharger 2 D[907]

;-----------------------------------------
;Revision 1.00 19/12/2005 D.J. First Issue
;-----------------------------------------

DischargerEnable 		= ((D[12] > 0) AND NOT Std.HaltSys)

;I_BagAtBuffer			= X[6].X07
I_OpenBag				= (CAN[2].DropLoad)
KEV         				= (CAN[2].DropLoad)
I_LoadDropped			= CAN[2].LoadDropped OR TestDropped
I_BagAtBuffer			= X[6].X09 OR TestBuffer
I_BagAtDischarger		= X[6].X10 OR TestAtDisch
I_BagEmpty			  	= TRUE

I_BagAtEmptyBuffer		= FALSE ;X[6].X13
O_EmptyBagBufferOpen	= FALSE ;Y[6].Y13

O_BagReady				= FALSE
O_OpenBuffer 			= FALSE
O_Steadys				= FALSE
O_Closer				= FALSE
O_OpenBag				= FALSE
O_OpenStop				= FALSE

Request.DC[2] 			= FALSE
Request.DCEmptyRelease[2] = FALSE
;Alarm
Alarm[7].Name 			= almNoAlarm ;Clear sequence alarm name
Alarm[7].Bag 			= 60
Alarm[7].Beacon			= TRUE
Alarm[7].Extra			= 0
Alarm[7].Time			= 3000

;Setup Sequence
STEP = D[907]
;Setup Pulse contact
PLS = (STEP <> LASTSTEP)
LASTSTEP = STEP

;Step 0 - Disabled
IF (STEP = 0) THEN
	;Disabled
ENDIF

;Check Status - Bag settled at buffer, no bag at discharger, bag at buffer on screen and no bag at discharger on the screen
TON_10ms(I_BagAtBuffer,300,SettledAtBuffer,SettledAtBufferET)
IF (STEP = 1) THEN
	IF (NOT I_BagAtDischarger AND  (Bag[60].Cat = 0) AND NOT Std.HaltSys AND DischargerEnable AND SettledAtBuffer) THEN
		Request.DC[2] = TRUE
		D[907] = 2
	ENDIF
	IF I_BagAtDischarger THEN
		;D[907] = 2
	ENDIF
	IF (Bag[60].Cat > 0) THEN
		Alarm[7].Name = almBagDataError
	ELSE IF I_BagAtDischarger THEN
		Alarm[7].Name = almSwitchFault
	ELSE IF (Bag[61].Cat > 0) AND NOT I_BagAtBuffer THEN
		Alarm[7].Name 	= almBagNotAtProx
		Alarm[7].Bag	= 61
	ELSE IF (Bag[61].Cat = 0) AND I_BagAtBuffer AND DischargerEnable  THEN
		Alarm[7].Name 	= almBagNotShownOnScreen
		Alarm[7].Bag	= 61
	ENDIF
ENDIF

;Wait for bag in discharger
IF (STEP = 2) THEN
	O_OpenBuffer 	= TRUE
	IF I_BagAtDischarger THEN
		D[907] = 3
	ENDIF
	Alarm[7].Name = almNoAlarm ;almBagNotArrived
ENDIF

;Let bag settle in discharger
TON_10ms(((STEP = 3) AND I_BagAtDischarger),1000,SettledAtDischarger,SettledAtDischargerET)
IF (STEP = 3) THEN
	IF (Bag[60].Cat = 0) AND (Bag[61].Cat > 0)  THEN
		Bag[60] = Bag[61]
		Bag[61] = Bag[0]
	ENDIF
	IF SettledAtDischarger THEN
		D[907] = 4
	ENDIF
	Alarm[7].Name = almBagNotSettled
ENDIF

IF (D[982] = 0) AND (STEP = 6) THEN
	IF (Bag[61].Cat>0) AND (Bag[60].Cat>0) AND (Bag[60].Cat = Bag[61].Cat) THEN
		D[982] = 2
	ELSE
		D[982] = 1
	ENDIF

ENDIF

IF (D[982] = 1) AND( (STEP = 6) OR (STEP = 7) OR (STEP = 8)) THEN
	CAN[2].LoadFinished = TRUE
ELSE
	CAN[2].LoadFinished = FALSE
ENDIF

;Allow steadys to move down
TON_10ms((STEP = 4),400,SteadysDown,SteadysDownET)
IF (STEP = 4) THEN
	IF SteadysDown AND( (Bag[61].Cat>0) OR (D[982] = 1)) THEN
		D[907] = 5
	ENDIF
	IF (Bag[60].Cat = Std.MaxCats) THEN
		D[907] = 8
	ENDIF
ENDIF

;Steady cylinders on from steps 4 - 9
O_Steadys = ((STEP >= 4) AND (STEP <= 9))

;Bag opener on from step 5 - 8
O_OpenBag = ((STEP >= 6) AND (STEP <= 8))

CodeStep  = ((STEP >= 4) AND (STEP <= 5))

;Wash Codes
IF CodeStep THEN

	Weight = Bag[60].Wgt

	;round up weight to give to wash machine
	Remainder = SINT(Bag[60].Wgt MOD 10)
	IF (Remainder > 4) THEN
		WgtRound = (Weight + 10)
	ELSE
		WgtRound = Weight
	ENDIF

	;WashCodes
	;if Below the Machine limit of 99 and no WashCode has been entered then send the Category

	CAN[2].Category 	= Bag[60].Cat
	CAN[2].Customer 	= Bag[60].Cus
	CAN[2].Weight   	= (WgtRound / 10) ;rounded up weight divide by 10
	;CAN[1].DoubleLoad 	= (Batch > 0)
ELSE
	CAN[2].Category 	= 0
	CAN[2].Customer 	= 0
	CAN[2].Weight   	= 0
	;CAN[1].DoubleLoad 	= FALSE

ENDIF

;Bag Ready to Washing Machine
IF (STEP = 5) THEN
	CAN[2].BagReady 		= TRUE

	IF I_OpenBag OR TestDischarger THEN
		D[907] = 6
	ENDIF
ELSE
	CAN[2].BagReady = FALSE
ENDIF

;Set LoadDropped to False
IF (STEP <> 6) THEN
	LoadDropped = FALSE
ENDIF

;Open Bag Until LoadDropped recieved and has been open for 6 seconds
TON_10ms((STEP = 6),600,MinOpen,MinOpenET) ;ET means Elapsed Time
TON_10ms((STEP = 6) AND NOT I_DischargerBagEmpty ,100,BagEmpty,BagEmptyET)

IF (STEP = 6) THEN

	IF I_LoadDropped  OR TestDischarger THEN

		LoadDropped = TRUE
	ENDIF

	IF (LoadDropped AND MinOpen) THEN
		;Write Report
		;------------

	ENDIF
	IF (LoadDropped AND MinOpen ) THEN
		IF (ReportUnloading[2].Cat = 0) THEN
			ReportUnloading[2].Cat = UINT(Bag[60].Cat)	;Category
			ReportUnloading[2].Cus = Bag[60].Cus		;Customer
			ReportUnloading[2].Wgt = Bag[60].Wgt		;Weight
			ReportUnloading[2].Cnt = 0					;Count
			ReportUnloading[2].Stn = 0					;Station
			ReportUnloading[2].Mcn = 2					;Machine
		ENDIF
		D[907] = 7
	ENDIF
	Alarm[7].Name = almLoadNotDropped
	ELSE
	LoadDropped = FALSE
ENDIF

;Change display to empty bag
IF (STEP = 7) THEN
	IF ((NOT I_OpenBag  AND I_BagEmpty) OR TestDrop) THEN
		Bag[60].Prg 	= Std.MaxProg
		Bag[60].Cat 	= Std.MaxCats
		Bag[60].Cus 	= Std.MaxCust

		D[907] 			= 8
	ENDIF
	Alarm[7].Name = almGeneralSequence
ENDIF

;Close bag
TON_10ms((STEP = 8),700,CloserDown,CloserDownET)
IF (STEP = 8) THEN
	O_Closer = TRUE
	IF CloserDown THEN
		D[907] = 9
	ENDIF
ENDIF

;Allow closer to go back up
TON_10ms((STEP = 9),700,CloserUp,CloserUpET)
IF (STEP = 9) THEN
		IF PLS THEN
		IF (D[982]>0) THEN
			D[982] = (D[982]-1)
		ENDIF
	ENDIF
	IF CloserUp THEN
		D[907] = 10
	ENDIF
ENDIF

;Allow steadys to go up
TON_10ms((STEP = 10),400,SteadyUp,SteadyUpET)
IF (STEP = 10) THEN
	IF SteadyUp THEN
		D[907] = 11
	ENDIF
ENDIF

;Request empty bag release
IF (STEP = 11) THEN

	IF Line[33].Clear THEN
		C[33]  = 0
		D[907] = 12
	ENDIF
ENDIF

;Open buffer stop - unitl bag out
IF (STEP = 12) THEN
	O_OpenStop = TRUE
	Bag[60].Cat = 0
	Bag[60].Cus = 0
	Bag[60].Wgt = 0
	IF Line[33].Trip THEN
		D[907] = 1
	ENDIF
	Alarm[7].Name = almBagNotReleased
ENDIF

;Alarms
TimerAlarm.IN 	= NOT PLS AND (Alarm[7].Name > 0)
TimerAlarm.PT 	= Alarm[7].Time
TimerAlarm FUB TON_10ms()
Alarm[7].On 	= TimerAlarm.Q
Alarm[7].ET 	= TimerAlarm.ET

;Outputs
Y[6].Y07 = O_OpenBuffer
Y[6].Y08 = O_Steadys
Y[6].Y09 = O_OpenBag
Y[6].Y11 = O_OpenStop
Y[6].Y10 = O_Closer
END_PROGRAM
```

### Program Logical/Sequences/10ms/8_sdc3 (IEC) - * SDC2 Machine 2 CAN

#### 7_sdc2.var
```iecst
VAR RETAIN
	STEP : UINT;
	PLS : BOOL;
	LASTSTEP : UINT;
	SteadyUp : BOOL;
	CloserUpET : TIME;
	SteadysDown : BOOL;
	SteadysDownET : TIME;
	LoadDropped : BOOL;
	SteadyUpET : TIME;
	CloserDownET : TIME;
	SettledAtDischargerET : TIME;
	MinOpenET : TIME;
	SettledAtDischarger : BOOL;
	CloserDown : BOOL;
	MinOpen : BOOL;
	CloserUp : BOOL;
	SettledAtBuffer : BOOL;
	SettledAtBufferET : TIME;
	I_BagAtBuffer : BOOL;
	O_OpenStop : BOOL;
	O_OpenBag : BOOL;
	O_Steadys : BOOL;
	O_OpenBuffer : BOOL;
	O_Closer : BOOL;
	I_BagAtDischarger : BOOL;
	I_OpenBag : BOOL;
	I_LoadDropped : BOOL;
	TestDrop : BOOL;
END_VAR
VAR
	DischargerEnable : BOOL;
	TestDischarger : BOOL;
	I_BagEmpty : BOOL;
	O_BagReady : BOOL;
	WgtRound : UINT;
	TimerAlarm : TON_10ms;
	I_BagReleased : BOOL;
	O_EmptyBagBufferOpen : BOOL;
	I_BagAtEmptyBuffer : BOOL;
	Remainder : UINT;
	CodeStep : BOOL;
	I_DischargerBagEmpty : BOOL;
	BagEmpty : BOOL;
	BagEmptyET : TIME;
	BCD_BIN_CAT : BCD_BIN_OUTPUT;
	BCD_BIN_CUS : BCD_BIN_OUTPUT;
	BCD_BIN_WGT : BCD_BIN_OUTPUT;
	TestDropped : BOOL;
	TestBuffer : BOOL;
	TestAtDisch : BOOL;
	Weight : UINT;
END_VAR
```

#### 7_sdc2Cyclic.ab
```automation-basic
PROGRAM _CYCLIC
	(* cyclic program *)

;Sequence 7 - Discharger 2 D[907]

;-----------------------------------------
;Revision 1.00 19/12/2005 D.J. First Issue
;-----------------------------------------

DischargerEnable 		= ((D[13] > 0) AND NOT Std.HaltSys)

;I_BagAtBuffer			= X[6].X07
I_OpenBag				= X[6].X16
;I_LoadDropped			= CAN[2].LoadDropped OR TestDropped
I_BagAtBuffer			= X[6].X13 OR TestBuffer
I_BagAtDischarger		= X[6].X14 OR TestAtDisch
I_BagEmpty			  	= FALSE
Request.DC[3]           = FALSE

I_BagAtEmptyBuffer		= FALSE ;X[6].X13
O_EmptyBagBufferOpen	= FALSE ;Y[6].Y13

O_BagReady				= FALSE
O_OpenBuffer 			= FALSE
O_Steadys				= FALSE
O_Closer				= FALSE
O_OpenBag				= FALSE
O_OpenStop				= FALSE
Request.DCEmptyRelease[3] = FALSE

;Alarm
Alarm[8].Name 			= almNoAlarm ;Clear sequence alarm name
Alarm[8].Bag 			= 70
Alarm[8].Beacon			= TRUE
Alarm[8].Extra			= 0
Alarm[8].Time			= 3000

;Setup Sequence
STEP = D[908]
;Setup Pulse contact
PLS = (STEP <> LASTSTEP)
LASTSTEP = STEP

;Step 0 - Disabled
IF (STEP = 0) THEN
	;Disabled
ENDIF

;Check Status - Bag settled at buffer, no bag at discharger, bag at buffer on screen and no bag at discharger on the screen
TON_10ms(I_BagAtBuffer,300,SettledAtBuffer,SettledAtBufferET)
IF (STEP = 1) THEN
	IF (NOT I_BagAtDischarger AND (Bag[71].Cat > 0) AND  (Bag[70].Cat = 0) AND NOT Std.HaltSys AND DischargerEnable AND SettledAtBuffer) THEN

		D[908] = 2
	ENDIF
	IF I_BagAtDischarger THEN
		;D[907] = 2
	ENDIF
	IF (Bag[70].Cat > 0) THEN
		Alarm[8].Name = almBagDataError
	ELSE IF I_BagAtDischarger THEN
		Alarm[8].Name = almSwitchFault
	ELSE IF (Bag[71].Cat > 0) AND NOT I_BagAtBuffer THEN
		Alarm[8].Name 	= almBagNotAtProx
		Alarm[8].Bag	= 71
	ELSE IF (Bag[71].Cat = 0) AND I_BagAtBuffer AND DischargerEnable  THEN
		Alarm[8].Name 	= almBagNotShownOnScreen
		Alarm[8].Bag	= 71
	ENDIF
ENDIF

;Wait for bag in discharger
IF (STEP = 2) THEN
	O_OpenBuffer 	= TRUE
	IF I_BagAtDischarger THEN
		D[908] = 3
	ENDIF
	Alarm[8].Name = almNoAlarm ;almBagNotArrived
ENDIF

;Let bag settle in discharger
TON_10ms(((STEP = 3) AND I_BagAtDischarger),1000,SettledAtDischarger,SettledAtDischargerET)
IF (STEP = 3) THEN
	IF (Bag[70].Cat = 0) AND (Bag[71].Cat > 0) THEN
		Bag[70] = Bag[71]
		Bag[71] = Bag[0]
	ENDIF
	IF SettledAtDischarger THEN
		D[908] = 4
	ENDIF
	Alarm[8].Name = almBagNotSettled
ENDIF

;Allow steadys to move down
TON_10ms((STEP = 4),400,SteadysDown,SteadysDownET)
IF (STEP = 4) THEN
	IF SteadysDown THEN
		D[908] = 5
	ENDIF
	IF (Bag[70].Cat = Std.MaxCats) THEN
		D[908] = 8
	ENDIF
ENDIF

;Steady cylinders on from steps 4 - 9
O_Steadys = ((STEP >= 4) AND (STEP <= 9))

;Bag opener on from step 5 - 8
O_OpenBag = ((STEP >= 6) AND (STEP <= 8))

;CodeStep  = ((STEP >= 4) AND (STEP <= 5))

;Wash Codes
IF CodeStep THEN

	Weight = Bag[70].Wgt

	;round up weight to give to wash machine
	Remainder = SINT(Bag[70].Wgt MOD 10)
	IF (Remainder > 4) THEN
		WgtRound = (Weight + 10)
	ELSE
		WgtRound = Weight
	ENDIF

ELSE

ENDIF

;Bag Ready to Washing Machine
IF (STEP = 5) THEN
	O_BagReady = TRUE
	IF I_OpenBag OR TestDischarger THEN
		D[908] = 6
	ENDIF
ELSE

ENDIF

;Set LoadDropped to False
IF (STEP <> 6) THEN
	LoadDropped = FALSE
ENDIF

;Open Bag Until LoadDropped recieved and has been open for 6 seconds
TON_10ms((STEP = 6),600,MinOpen,MinOpenET) ;ET means Elapsed Time
TON_10ms((STEP = 6) AND NOT I_DischargerBagEmpty ,100,BagEmpty,BagEmptyET)

IF (STEP = 6) THEN

		LoadDropped = TRUE

	IF (LoadDropped AND MinOpen) THEN
		;Write Report
		;------------

	ENDIF
	IF (LoadDropped AND MinOpen ) THEN
		IF (ReportUnloading[3].Cat = 0) THEN
			ReportUnloading[3].Cat = UINT(Bag[70].Cat)	;Category
			ReportUnloading[3].Cus = Bag[70].Cus		;Customer
			ReportUnloading[3].Wgt = Bag[70].Wgt		;Weight
			ReportUnloading[3].Cnt = 0					;Count
			ReportUnloading[3].Stn = 0					;Station
			ReportUnloading[3].Mcn = 3					;Machine
		ENDIF
		D[908] = 7
	ENDIF
	Alarm[8].Name = almLoadNotDropped
	ELSE
	LoadDropped = FALSE
ENDIF

;Change display to empty bag
IF (STEP = 7) THEN
	O_BagReady = Std.Clock500ms
	IF (( I_OpenBag ) OR TestDrop) THEN
		Bag[70].Prg 	= Std.MaxProg
		Bag[70].Cat 	= Std.MaxCats
		Bag[70].Cus 	= Std.MaxCust

		D[908] 			= 8
	ENDIF
	Alarm[8].Name = almGeneralSequence
ENDIF

;Close bag
TON_10ms((STEP = 8),700,CloserDown,CloserDownET)
IF (STEP = 8) THEN
	O_Closer = TRUE
	IF CloserDown THEN
		D[908] = 9
	ENDIF
ENDIF

;Allow closer to go back up
TON_10ms((STEP = 9),700,CloserUp,CloserUpET)
IF (STEP = 9) THEN
	IF CloserUp THEN
		D[908] = 10
	ENDIF
ENDIF

;Allow steadys to go up
TON_10ms((STEP = 10),400,SteadyUp,SteadyUpET)
IF (STEP = 10) THEN
	IF SteadyUp THEN
		D[908] = 11
	ENDIF
ENDIF

;Request empty bag release
IF (STEP = 11) THEN
	Request.DCEmptyRelease[3] = TRUE
	;Request.DC[3] = TRUE
	IF Enable.DCEmptyRelease[3] THEN
		;C[32]  = 0
		D[908] = 12
	ENDIF
ENDIF

;Open buffer stop - unitl bag out
IF (STEP = 12) THEN
	O_OpenStop = TRUE
	Bag[70].Cat = 0
	Bag[70].Cus = 0
	Bag[70].Wgt = 0
	IF NOT Enable.DCEmptyRelease[3] THEN
		D[908] = 1
	ENDIF
	Alarm[8].Name = almBagNotReleased
ENDIF

;Alarms
TimerAlarm.IN 	= NOT PLS AND (Alarm[8].Name > 0)
TimerAlarm.PT 	= Alarm[8].Time
TimerAlarm FUB TON_10ms()
Alarm[8].On 	= TimerAlarm.Q
Alarm[8].ET 	= TimerAlarm.ET

;Outputs
Y[6].Y13 = O_OpenBuffer
Y[6].Y14 = O_Steadys
Y[6].Y15 = O_OpenBag
Y[7].Y01 = O_OpenStop
Y[6].Y16 = O_Closer
Y[7].Y02 = O_BagReady
END_PROGRAM
```

### Program Logical/Sequences/10ms/9_sdc4 (IEC) - * SDC2 Machine 2 CAN

#### 7_sdc2.var
```iecst
VAR RETAIN
	STEP : UINT;
	PLS : BOOL;
	LASTSTEP : UINT;
	SteadyUp : BOOL;
	CloserUpET : TIME;
	SteadysDown : BOOL;
	SteadysDownET : TIME;
	LoadDropped : BOOL;
	SteadyUpET : TIME;
	CloserDownET : TIME;
	SettledAtDischargerET : TIME;
	MinOpenET : TIME;
	SettledAtDischarger : BOOL;
	CloserDown : BOOL;
	MinOpen : BOOL;
	CloserUp : BOOL;
	SettledAtBuffer : BOOL;
	SettledAtBufferET : TIME;
	I_BagAtBuffer : BOOL;
	O_OpenStop : BOOL;
	O_OpenBag : BOOL;
	O_Steadys : BOOL;
	O_OpenBuffer : BOOL;
	O_Closer : BOOL;
	I_BagAtDischarger : BOOL;
	I_OpenBag : BOOL;
	I_LoadDropped : BOOL;
	TestDrop : BOOL;
END_VAR
VAR
	DischargerEnable : BOOL;
	TestDischarger : BOOL;
	I_BagEmpty : BOOL;
	O_BagReady : BOOL;
	WgtRound : UINT;
	TimerAlarm : TON_10ms;
	I_BagReleased : BOOL;
	O_EmptyBagBufferOpen : BOOL;
	I_BagAtEmptyBuffer : BOOL;
	Remainder : UINT;
	CodeStep : BOOL;
	I_DischargerBagEmpty : BOOL;
	BagEmpty : BOOL;
	BagEmptyET : TIME;
	BCD_BIN_CAT : BCD_BIN_OUTPUT;
	BCD_BIN_CUS : BCD_BIN_OUTPUT;
	BCD_BIN_WGT : BCD_BIN_OUTPUT;
	TestDropped : BOOL;
	TestBuffer : BOOL;
	TestAtDisch : BOOL;
	Weight : UINT;
	kev : INT;
END_VAR
```

#### 7_sdc2Cyclic.ab
```automation-basic
PROGRAM _CYCLIC
	(* cyclic program *)

;Sequence 7 - Discharger 2 D[907]

;-----------------------------------------
;Revision 1.00 19/12/2005 D.J. First Issue
;-----------------------------------------

DischargerEnable 		= ((D[14] > 0) AND NOT Std.HaltSys)

;I_BagAtBuffer			= X[6].X07
I_OpenBag				= X[7].X04 ;[2].DropLoad OR TestDrop
I_LoadDropped			= CAN[2].LoadDropped OR TestDropped
I_BagAtBuffer			= X[7].X01 OR TestBuffer
I_BagAtDischarger		= X[7].X02 OR TestAtDisch
I_BagEmpty			  	= TRUE

I_BagAtEmptyBuffer		= FALSE ;X[6].X13
O_EmptyBagBufferOpen	= FALSE ;Y[6].Y13
EnableRel.IC[1] 	    = FALSE

O_BagReady				= FALSE
O_OpenBuffer 			= FALSE
O_Steadys				= FALSE
O_Closer				= FALSE
O_OpenBag				= FALSE
O_OpenStop				= FALSE

;Request.DC[2] 			= FALSE
;Request.DCEmptyRelease[2] = FALSE
;Alarm
Alarm[9].Name 			= almNoAlarm ;Clear sequence alarm name
Alarm[9].Bag 			= 75
Alarm[9].Beacon			= TRUE
Alarm[9].Extra			= 0
Alarm[9].Time			= 3000

;Setup Sequence
STEP = D[909]
;Setup Pulse contact
PLS = (STEP <> LASTSTEP)
LASTSTEP = STEP

;Step 0 - Disabled
IF (STEP = 0) THEN
	;Disabled
ENDIF

;Check Status - Bag settled at buffer, no bag at discharger, bag at buffer on screen and no bag at discharger on the screen
TON_10ms(I_BagAtBuffer,300,SettledAtBuffer,SettledAtBufferET)
IF (STEP = 1) THEN
	IF (NOT I_BagAtDischarger AND  (Bag[75].Cat = 0) AND NOT Std.HaltSys AND DischargerEnable AND RequestRel.IC[1]) THEN
		;Request.DC[2] = TRUE
		D[909] = 2
	ENDIF
	IF (NOT I_BagAtDischarger AND  (Bag[75].Cat = 0) AND NOT Std.HaltSys AND DischargerEnable ) THEN
		;Request.DC[2] = TRUE
		kev = 2
	ENDIF
	IF I_BagAtDischarger THEN
		;D[907] = 2
	ENDIF
	IF (Bag[188].Cat > 0) THEN
		Alarm[9].Name = almBagDataError
	ELSE IF I_BagAtDischarger THEN
		Alarm[9].Name = almSwitchFault
	ELSE IF (Bag[75].Cat > 0) AND NOT I_BagAtBuffer THEN
		Alarm[9].Name 	= almBagNotAtProx
		Alarm[9].Bag	= 75
	ELSE IF (Bag[75].Cat = 0) AND I_BagAtBuffer AND DischargerEnable  THEN
		Alarm[9].Name 	= almBagNotShownOnScreen
		Alarm[9].Bag	= 75
	ENDIF
ENDIF

;Wait for bag in discharger
IF (STEP = 2) THEN
	EnableRel.IC[1] 	= TRUE
	IF I_BagAtDischarger THEN
		D[909] = 3
	ENDIF
	Alarm[9].Name = almNoAlarm ;almBagNotArrived
ENDIF

;Let bag settle in discharger
TON_10ms(((STEP = 3) AND I_BagAtDischarger),1000,SettledAtDischarger,SettledAtDischargerET)
IF (STEP = 3) THEN
	IF (Bag[75].Cat = 0) AND (Bag[76].Cat > 0) THEN
		Bag[75] = Bag[76]
		Bag[76] = Bag[0]
	ENDIF
	IF SettledAtDischarger THEN
		D[909] = 4
	ENDIF
	Alarm[9].Name = almBagNotSettled
ENDIF

;Allow steadys to move down
TON_10ms((STEP = 4),400,SteadysDown,SteadysDownET)
IF (STEP = 4) THEN
	IF SteadysDown THEN
		D[909] = 5
	ENDIF
	IF (Bag[75].Cat = Std.MaxCats) THEN
		D[909] = 8
	ENDIF
ENDIF

;Steady cylinders on from steps 4 - 9
O_Steadys = ((STEP >= 4) AND (STEP <= 9))

;Bag opener on from step 5 - 8
O_OpenBag = ((STEP >= 6) AND (STEP <= 8))

CodeStep  = ((STEP >= 4) AND (STEP <= 5))

;Wash Codes
IF CodeStep THEN

	Weight = Bag[75].Wgt

	;round up weight to give to wash machine
	Remainder = SINT(Bag[75].Wgt MOD 10)
	IF (Remainder > 4) THEN
		WgtRound = (Weight + 10)
	ELSE
		WgtRound = Weight
	ENDIF

	;WashCodes
	;if Below the Machine limit of 99 and no WashCode has been entered then send the Category
		;CAN[1].DoubleLoad 	= (Batch > 0)
ELSE
		;CAN[1].DoubleLoad 	= FALSE

ENDIF

;Bag Ready to Washing Machine
IF (STEP = 5) THEN
	O_BagReady = TRUE

	IF I_OpenBag OR TestDischarger THEN
		D[909] = 6
	ENDIF
ELSE

ENDIF

;Set LoadDropped to False
IF (STEP <> 6) THEN
	LoadDropped = FALSE
ENDIF

;Open Bag Until LoadDropped recieved and has been open for 6 seconds
TON_10ms((STEP = 6),600,MinOpen,MinOpenET) ;ET means Elapsed Time
TON_10ms((STEP = 6) AND NOT I_DischargerBagEmpty ,100,BagEmpty,BagEmptyET)

IF (STEP = 6) THEN

	;IF I_LoadDropped  OR TestDischarger THEN

		LoadDropped = TRUE
	;ENDIF

	IF (LoadDropped AND MinOpen) THEN
		;Write Report
		;------------

	ENDIF
	IF (LoadDropped AND MinOpen ) THEN
		IF (ReportUnloading[4].Cat = 0) THEN
			ReportUnloading[4].Cat = UINT(Bag[75].Cat)	;Category
			ReportUnloading[4].Cus = Bag[75].Cus		;Customer
			ReportUnloading[4].Wgt = Bag[75].Wgt		;Weight
			ReportUnloading[4].Cnt = 0					;Count
			ReportUnloading[4].Stn = 0					;Station
			ReportUnloading[4].Mcn = 4					;Machine
		ENDIF
		D[909] = 7
	ENDIF
	Alarm[9].Name = almLoadNotDropped
	ELSE
	LoadDropped = FALSE
ENDIF

;Change display to empty bag
IF (STEP = 7) THEN
	O_BagReady = Std.Clock100ms
	IF ((I_OpenBag) OR TestDrop) THEN
		Bag[75].Prg 	= Std.MaxProg
		Bag[75].Cat 	= Std.MaxCats
		Bag[75].Cus 	= Std.MaxCust

		D[909] 			= 8
	ENDIF
	Alarm[9].Name = almGeneralSequence
ENDIF

;Close bag
TON_10ms((STEP = 8),700,CloserDown,CloserDownET)
IF (STEP = 8) THEN
	O_Closer = TRUE
	IF CloserDown THEN
		D[909] = 9
	ENDIF
ENDIF

;Allow closer to go back up
TON_10ms((STEP = 9),700,CloserUp,CloserUpET)
IF (STEP = 9) THEN
	IF CloserUp THEN
		D[909] = 10
	ENDIF
ENDIF

;Allow steadys to go up
TON_10ms((STEP = 10),400,SteadyUp,SteadyUpET)
IF (STEP = 10) THEN
	IF SteadyUp THEN
		D[909] = 11
	ENDIF
ENDIF

;Request empty bag release
IF (STEP = 11) THEN
	;Request.DCEmptyRelease[2] = TRUE
	IF Line[45].Clear THEN
		C[45]  = 0
		D[909] = 12
	ENDIF
ENDIF

;Open buffer stop - unitl bag out
IF (STEP = 12) THEN
	O_OpenStop = TRUE
	Bag[75].Cat = 0
	Bag[75].Cus = 0
	Bag[75].Wgt = 0
	IF Line[45].Trip THEN
		D[909] = 1
	ENDIF
	Alarm[9].Name = almBagNotReleased
ENDIF

;Alarms
TimerAlarm.IN 	= NOT PLS AND (Alarm[9].Name > 0)
TimerAlarm.PT 	= Alarm[9].Time
TimerAlarm FUB TON_10ms()
Alarm[9].On 	= TimerAlarm.Q
Alarm[9].ET 	= TimerAlarm.ET

;Outputs
;Y[6].Y06 = O_OpenBuffer
Y[7].Y04 = O_Steadys
Y[7].Y05 = O_OpenBag
Y[7].Y07 = O_OpenStop
Y[7].Y06 = O_Closer
Y[7].Y08 = O_BagReady
END_PROGRAM
```

### Program Logical/Sequences/10ms/10_sdc5 (IEC) - * SDC2 Machine 2 CAN
